C03605=1052.364,227.294,-95.651,172.051,36.072,156.780
C03606=1052.357,227.046,-95.623,172.050,36.069,156.779
C03607=1052.351,226.797,-95.597,172.047,36.065,156.779
C03608=1052.344,226.549,-95.569,172.045,36.062,156.778
C03609=1052.337,226.300,-95.542,172.042,36.058,156.777
C03610=1052.331,226.052,-95.515,172.040,36.055,156.777
C03611=1052.325,225.803,-95.488,172.038,36.052,156.776
C03612=1052.318,225.555,-95.460,172.036,36.048,156.775
C03613=1052.312,225.307,-95.434,172.034,36.045,156.775
C03614=1052.306,225.058,-95.406,172.032,36.042,156.774
C03615=1052.300,224.810,-95.379,172.029,36.038,156.773
C03616=1052.294,224.561,-95.352,172.027,36.035,156.772
C03617=1052.287,224.313,-95.326,172.026,36.032,156.772
C03618=1052.280,224.064,-95.299,172.023,36.028,156.771
C03619=1052.274,223.816,-95.271,172.021,36.024,156.770
C03620=1052.268,223.567,-95.244,172.018,36.021,156.770
C03621=1052.261,223.318,-95.217,172.016,36.018,156.769
C03622=1052.255,223.071,-95.190,172.015,36.014,156.768
C03623=1052.249,222.821,-95.163,172.012,36.011,156.768
C03624=1052.243,222.573,-95.137,172.010,36.007,156.767
C03625=1052.236,222.325,-95.109,172.008,36.004,156.766
C03626=1052.230,222.077,-95.082,172.005,36.000,156.765
C03627=1052.224,221.828,-95.055,172.004,35.997,156.765
C03628=1052.218,221.580,-95.028,172.001,35.993,156.764
C03629=1052.211,221.328,-95.001,171.999,35.990,156.763
C03630=1052.205,221.076,-94.974,171.997,35.987,156.763
C03631=1052.198,220.824,-94.946,171.995,35.983,156.762
C03632=1052.192,220.572,-94.919,171.993,35.979,156.761
C03633=1052.185,220.323,-94.893,171.991,35.976,156.760
C03634=1052.179,220.075,-94.865,171.988,35.973,156.760
C03635=1052.173,219.827,-94.839,171.987,35.969,156.759
C03636=1052.166,219.578,-94.812,171.985,35.966,156.758
C03637=1052.160,219.330,-94.786,171.982,35.963,156.758
C03638=1052.153,219.081,-94.759,171.980,35.959,156.757
C03639=1052.147,218.832,-94.733,171.977,35.956,156.756
C03640=1052.140,218.584,-94.706,171.976,35.953,156.756
C03641=1052.134,218.336,-94.679,171.974,35.949,156.755
C03642=1052.128,218.087,-94.652,171.971,35.945,156.754
C03643=1052.121,217.839,-94.626,171.970,35.942,156.753
C03644=1052.115,217.590,-94.599,171.968,35.939,156.753
C03645=1052.108,217.342,-94.573,171.965,35.935,156.752
C03646=1052.102,217.093,-94.546,171.963,35.932,156.751
C03647=1052.096,216.844,-94.519,171.962,35.929,156.751
C03648=1052.089,216.596,-94.493,171.959,35.925,156.750
C03649=1052.083,216.347,-94.466,171.957,35.921,156.749
C03650=1052.077,216.099,-94.440,171.955,35.918,156.749
C03651=1052.070,215.850,-94.413,171.953,35.915,156.748
C03652=1052.064,215.602,-94.387,171.951,35.911,156.747
C03653=1052.057,215.353,-94.360,171.949,35.908,156.746
C03654=1052.051,215.105,-94.334,171.947,35.904,156.746
C03655=1052.045,214.857,-94.307,171.945,35.900,156.745
C03656=1052.039,214.608,-94.280,171.942,35.897,156.744
C03657=1052.032,214.359,-94.254,171.941,35.894,156.744
C03658=1052.026,214.111,-94.227,171.939,35.890,156.743
C03659=1052.019,213.862,-94.201,171.936,35.887,156.742
C03660=1052.013,213.614,-94.174,171.934,35.883,156.741
C03661=1052.007,213.365,-94.149,171.933,35.880,156.741
C03662=1052.001,213.116,-94.122,171.930,35.876,156.740
C03663=1051.994,212.868,-94.096,171.928,35.873,156.739
C03664=1051.988,212.619,-94.069,171.927,35.869,156.739
C03665=1051.982,212.371,-94.043,171.924,35.865,156.738
C03666=1051.976,212.123,-94.016,171.922,35.862,156.737
C03667=1051.969,211.874,-93.990,171.921,35.859,156.737
C03668=1051.963,211.625,-93.964,171.918,35.855,156.736
C03669=1051.957,211.377,-93.938,171.916,35.852,156.735
C03670=1051.950,211.128,-93.911,171.914,35.848,156.734
C03671=1051.944,210.880,-93.885,171.912,35.845,156.734
C03672=1051.938,210.631,-93.859,171.910,35.841,156.733
C03673=1051.930,210.382,-93.833,171.908,35.838,156.732
C03674=1051.925,210.134,-93.806,171.906,35.834,156.732
C03675=1051.918,209.886,-93.780,171.905,35.831,156.731
C03676=1051.911,209.637,-93.755,171.902,35.828,156.730
C03677=1051.906,209.388,-93.728,171.900,35.824,156.730
C03678=1051.899,209.140,-93.702,171.899,35.820,156.729
C03679=1051.892,208.891,-93.676,171.896,35.817,156.728
C03680=1051.886,208.643,-93.650,171.894,35.813,156.727
C03681=1051.881,208.395,-93.624,171.893,35.810,156.727
C03682=1051.873,208.148,-93.598,171.890,35.807,156.726
C03683=1051.867,207.901,-93.572,171.888,35.803,156.725
C03684=1051.861,207.653,-93.546,171.887,35.799,156.725
C03685=1051.855,207.405,-93.520,171.884,35.796,156.724
C03686=1051.848,207.157,-93.494,171.883,35.793,156.723
C03687=1051.842,206.910,-93.469,171.881,35.789,156.722
C03688=1051.835,206.663,-93.442,171.878,35.785,156.722
C03689=1051.810,205.611,-93.337,171.657,35.690,156.704
C03690=1051.803,205.363,-93.312,171.654,35.688,156.704
C03691=1051.797,205.114,-93.287,171.652,35.686,156.703
C03692=1051.791,204.865,-93.262,171.649,35.683,156.703
C03693=1051.786,204.617,-93.237,171.647,35.680,156.702
C03694=1051.779,204.368,-93.212,171.644,35.678,156.702
C03695=1051.774,204.119,-93.187,171.642,35.675,156.701
C03696=1051.767,203.870,-93.162,171.639,35.672,156.701
C03697=1051.762,203.621,-93.138,171.637,35.669,156.700
C03698=1051.756,203.373,-93.112,171.634,35.667,156.699
C03699=1051.750,203.124,-93.087,171.632,35.664,156.699
C03700=1051.744,202.876,-93.063,171.629,35.661,156.698
C03701=1051.737,202.627,-93.038,171.626,35.659,156.698
C03702=1051.732,202.378,-93.013,171.624,35.656,156.697
C03703=1051.725,202.129,-92.988,171.622,35.653,156.697
C03704=1051.720,201.881,-92.964,171.619,35.651,156.696
C03705=1051.714,201.632,-92.938,171.617,35.648,156.696
C03706=1051.708,201.383,-92.914,171.614,35.645,156.695
C03707=1051.702,201.135,-92.889,171.612,35.643,156.695
C03708=1051.696,200.886,-92.865,171.609,35.640,156.694
C03709=1051.689,200.637,-92.840,171.606,35.638,156.694
C03710=1051.683,200.388,-92.815,171.604,35.635,156.693
C03711=1051.678,200.140,-92.791,171.602,35.633,156.693
C03712=1051.671,199.891,-92.766,171.600,35.630,156.692
C03713=1051.665,199.642,-92.742,171.596,35.627,156.692
C03714=1051.658,199.394,-92.717,171.594,35.625,156.691
C03715=1051.652,199.145,-92.693,171.592,35.622,156.691
C03716=1051.647,198.896,-92.668,171.590,35.620,156.690
C03717=1051.640,198.648,-92.644,171.586,35.617,156.690
C03718=1051.634,198.399,-92.619,171.584,35.614,156.689
C03719=1051.628,198.150,-92.595,171.582,35.612,156.689
C03720=1051.622,197.902,-92.570,171.580,35.610,156.688
C03721=1051.615,197.653,-92.546,171.578,35.607,156.688
C03722=1051.610,197.403,-92.521,171.574,35.605,156.687
C03723=1051.604,197.155,-92.497,171.572,35.602,156.687
C03724=1051.597,196.907,-92.472,171.570,35.600,156.687
C03725=1051.591,196.657,-92.448,171.568,35.597,156.686
C03726=1051.585,196.409,-92.424,171.564,35.594,156.685
C03727=1051.579,196.160,-92.400,171.562,35.592,156.685
C03728=1051.573,195.912,-92.375,171.560,35.589,156.684
C03729=1051.567,195.663,-92.351,171.558,35.587,156.684
C03730=1051.561,195.414,-92.326,171.556,35.584,156.684
C03731=1051.555,195.165,-92.302,171.552,35.582,156.683
C03732=1051.549,194.916,-92.278,171.550,35.579,156.683
C03733=1051.543,194.668,-92.253,171.548,35.577,156.682
C03734=1051.537,194.419,-92.229,171.546,35.574,156.682
C03735=1051.531,194.171,-92.205,171.543,35.571,156.681
C03736=1051.525,193.921,-92.180,171.541,35.569,156.681
C03737=1051.519,193.672,-92.156,171.538,35.566,156.680
C03738=1051.513,193.424,-92.132,171.536,35.564,156.680
C03739=1051.507,193.175,-92.108,171.534,35.562,156.679
C03740=1051.501,192.926,-92.084,171.531,35.559,156.679
C03741=1051.495,192.677,-92.060,171.529,35.557,156.678
C03742=1051.489,192.429,-92.035,171.527,35.554,156.678
C03743=1051.482,192.180,-92.011,171.524,35.552,156.677
C03744=1051.477,191.932,-91.986,171.522,35.549,156.677
C03745=1051.470,191.683,-91.962,171.519,35.547,156.676
C03746=1051.465,191.434,-91.938,171.517,35.544,156.676
C03747=1051.459,191.185,-91.914,171.515,35.542,156.675
C03748=1051.453,190.937,-91.890,171.513,35.539,156.675
C03749=1051.447,190.688,-91.866,171.509,35.536,156.674
C03750=1051.441,190.403,-91.838,171.507,35.534,156.674
C03751=1051.434,190.119,-91.810,171.505,35.531,156.673
C03752=1051.427,189.835,-91.783,171.502,35.528,156.673
C03753=1051.420,189.550,-91.756,171.500,35.525,156.672
C03754=1051.414,189.302,-91.732,171.497,35.523,156.672
C03755=1051.409,189.053,-91.708,171.494,35.520,156.671
C03756=1051.402,188.804,-91.684,171.492,35.518,156.671
C03757=1051.397,188.556,-91.660,171.490,35.515,156.670
C03758=1051.390,188.307,-91.636,171.487,35.513,156.670
C03759=1051.385,188.058,-91.611,171.485,35.510,156.669
C03760=1051.379,187.810,-91.588,171.483,35.508,156.669
C03761=1051.373,187.560,-91.563,171.481,35.505,156.668
C03762=1051.367,187.312,-91.540,171.479,35.502,156.668
C03763=1051.361,187.062,-91.516,171.476,35.500,156.667
C03764=1051.355,186.814,-91.492,171.473,35.497,156.667
C03765=1051.350,186.565,-91.468,171.471,35.495,156.666
C03766=1051.343,186.316,-91.444,171.469,35.492,156.666
C03767=1051.338,186.068,-91.419,171.467,35.490,156.665
C03768=1051.332,185.819,-91.396,171.464,35.487,156.665
C03769=1051.326,185.570,-91.372,171.462,35.485,156.665
C03770=1051.320,185.321,-91.348,171.460,35.483,156.664
C03771=1051.314,185.073,-91.324,171.458,35.480,156.664
C03772=1051.309,184.823,-91.301,171.456,35.478,156.663
C03773=1051.303,184.575,-91.277,171.453,35.475,156.663
C03774=1051.297,184.326,-91.253,171.451,35.473,156.662
C03775=1051.291,184.077,-91.229,171.449,35.470,156.662
C03776=1051.285,183.828,-91.206,171.446,35.468,156.661
C03777=1051.279,183.580,-91.182,171.444,35.466,156.661
C03778=1051.273,183.331,-91.159,171.441,35.463,156.660
C03779=1051.267,183.082,-91.135,171.439,35.461,156.660
C03780=1051.260,182.833,-91.111,171.437,35.458,156.659
C03781=1051.254,182.584,-91.088,171.435,35.457,156.659
C03782=1051.248,182.335,-91.064,171.433,35.454,156.659
C03783=1051.242,182.086,-91.041,171.430,35.452,156.658
C03784=1051.236,181.838,-91.017,171.428,35.450,156.658
C03785=1051.229,181.589,-90.994,171.425,35.447,156.657
C03786=1051.223,181.340,-90.970,171.423,35.445,156.657
C03787=1051.217,181.092,-90.948,171.421,35.442,156.656
C03788=1051.210,180.843,-90.924,171.419,35.440,156.656
C03789=1051.205,180.594,-90.901,171.416,35.438,156.656
C03790=1051.198,180.345,-90.877,171.414,35.435,156.655
C03791=1051.192,180.096,-90.854,171.412,35.434,156.655
C03792=1051.186,179.848,-90.830,171.410,35.431,156.654
C03793=1051.180,179.598,-90.807,171.408,35.429,156.654
C03794=1051.174,179.350,-90.783,171.405,35.426,156.653
C03795=1051.168,179.101,-90.761,171.403,35.424,156.653
C03796=1051.162,178.851,-90.737,171.401,35.422,156.653
C03797=1051.156,178.603,-90.714,171.399,35.419,156.652
C03798=1051.150,178.354,-90.691,171.396,35.417,156.652
C03799=1051.143,178.106,-90.667,171.394,35.415,156.651
C03800=1051.137,177.857,-90.644,171.391,35.412,156.651
C03801=1051.131,177.608,-90.621,171.389,35.411,156.650
C03802=1051.125,177.359,-90.598,171.387,35.408,156.650
C03803=1051.119,177.110,-90.574,171.385,35.406,156.649
C03804=1051.113,176.861,-90.551,171.383,35.404,156.649
C03805=1051.107,176.613,-90.528,171.380,35.401,156.649
C03806=1051.101,176.364,-90.505,171.378,35.399,156.648
C03807=1051.095,176.114,-90.481,171.376,35.396,156.648
C03808=1051.088,175.866,-90.458,171.374,35.394,156.647
C03809=1051.082,175.617,-90.435,171.372,35.392,156.647
C03810=1051.077,175.368,-90.413,171.370,35.389,156.646
C03811=1051.070,175.119,-90.389,171.367,35.388,156.646
C03812=1051.064,174.871,-90.366,171.365,35.385,156.646
C03813=1051.059,174.622,-90.343,171.363,35.383,156.645
C03814=1051.051,174.336,-90.317,171.361,35.380,156.645
C03815=1051.045,174.052,-90.290,171.358,35.378,156.644
C03816=1051.038,173.768,-90.264,171.355,35.375,156.644
C03817=1051.031,173.482,-90.237,171.353,35.372,156.643
C03818=1051.025,173.234,-90.214,171.351,35.370,156.643
C03819=1051.019,172.985,-90.191,171.349,35.368,156.642
C03820=1051.013,172.737,-90.168,171.347,35.365,156.642
C03821=1051.007,172.488,-90.145,171.344,35.363,156.642
C03822=1051.001,172.238,-90.122,171.342,35.361,156.641
C03823=1050.995,171.990,-90.098,171.340,35.358,156.641
C03824=1050.989,171.741,-90.075,171.338,35.357,156.640
C03825=1050.983,171.492,-90.052,171.336,35.354,156.640
C03826=1050.977,171.244,-90.030,171.334,35.352,156.639
C03827=1050.971,170.995,-90.007,171.331,35.350,156.639
C03828=1050.965,170.746,-89.984,171.329,35.347,156.639
C03829=1050.959,170.496,-89.961,171.327,35.345,156.638
C03830=1050.953,170.247,-89.938,171.325,35.343,156.638
C03831=1050.948,169.998,-89.915,171.323,35.340,156.637
C03832=1050.941,169.750,-89.893,171.321,35.338,156.637
C03833=1050.935,169.501,-89.870,171.318,35.336,156.636
C03834=1050.929,169.253,-89.846,171.316,35.333,156.636
C03835=1050.924,169.004,-89.823,171.314,35.331,156.635
C03836=1050.918,168.755,-89.800,171.312,35.329,156.635
C03837=1050.912,168.506,-89.777,171.310,35.327,156.635
C03838=1050.906,168.257,-89.755,171.307,35.324,156.634
C03839=1050.900,168.008,-89.732,171.305,35.322,156.634
C03840=1050.894,167.759,-89.709,171.303,35.320,156.633
C03841=1050.888,167.510,-89.686,171.301,35.317,156.633
C03842=1050.882,167.261,-89.663,171.299,35.315,156.633
C03843=1050.876,167.012,-89.641,171.297,35.313,156.632
C03844=1050.870,166.763,-89.618,171.294,35.310,156.632
C03845=1050.864,166.514,-89.595,171.292,35.309,156.631
C03846=1050.859,166.265,-89.572,171.291,35.306,156.631
C03847=1050.853,166.016,-89.549,171.289,35.304,156.630
C03848=1050.847,165.768,-89.527,171.287,35.302,156.630
C03849=1050.841,165.519,-89.504,171.285,35.299,156.630
C03850=1050.835,165.270,-89.481,171.282,35.297,156.629
C03851=1050.829,165.021,-89.458,171.280,35.295,156.629
C03852=1050.823,164.772,-89.436,171.278,35.292,156.628
C03853=1050.817,164.523,-89.413,171.276,35.290,156.628
C03854=1050.812,164.274,-89.391,171.274,35.288,156.627
C03855=1050.806,164.025,-89.368,171.272,35.285,156.627
C03856=1050.800,163.776,-89.345,171.269,35.283,156.627
C03857=1050.794,163.528,-89.322,171.267,35.281,156.626
C03858=1050.788,163.279,-89.299,171.265,35.279,156.626
C03859=1050.783,163.030,-89.277,171.264,35.276,156.625
C03860=1050.778,162.781,-89.255,171.262,35.274,156.625
C03861=1050.771,162.532,-89.232,171.260,35.272,156.624
C03862=1050.765,162.283,-89.209,171.257,35.269,156.624
C03863=1050.760,162.035,-89.186,171.255,35.267,156.624
C03864=1050.754,161.785,-89.164,171.253,35.265,156.623
C03865=1050.748,161.536,-89.142,171.251,35.263,156.623
C03866=1050.742,161.288,-89.119,171.249,35.260,156.622
C03867=1050.736,161.039,-89.096,171.247,35.258,156.622
C03868=1050.731,160.789,-89.074,171.245,35.256,156.622
C03869=1050.724,160.541,-89.051,171.243,35.254,156.621
C03870=1050.719,160.292,-89.028,171.241,35.252,156.621
C03871=1050.712,160.042,-89.007,171.239,35.249,156.620
C03872=1050.707,159.794,-88.984,171.237,35.247,156.620
C03873=1050.701,159.544,-88.962,171.235,35.245,156.619
C03874=1050.694,159.296,-88.940,171.232,35.243,156.619
C03875=1050.688,159.047,-88.917,171.230,35.240,156.619
C03876=1050.682,158.798,-88.895,171.228,35.239,156.618
C03877=1050.676,158.549,-88.873,171.226,35.236,156.618
C03878=1050.670,158.264,-88.847,171.224,35.234,156.617
C03879=1050.663,157.979,-88.822,171.222,35.231,156.617
C03880=1050.656,157.693,-88.796,171.219,35.229,156.616
C03881=1050.649,157.408,-88.771,171.217,35.227,156.616
C03882=1050.643,157.160,-88.749,171.215,35.224,156.616
C03883=1050.636,156.911,-88.727,171.213,35.222,156.615
C03884=1050.631,156.662,-88.704,171.211,35.220,156.615
C03885=1050.624,156.413,-88.682,171.209,35.218,156.614
C03886=1050.619,156.164,-88.660,171.207,35.215,156.614
C03887=1050.613,155.914,-88.638,171.204,35.214,156.614
C03888=1050.607,155.667,-88.616,171.202,35.211,156.613
C03889=1050.602,155.417,-88.594,171.201,35.209,156.613
C03890=1050.595,155.168,-88.572,171.199,35.207,156.612
C03891=1050.589,154.919,-88.550,171.197,35.205,156.612
C03892=1050.583,154.670,-88.527,171.195,35.203,156.612
C03893=1050.577,154.421,-88.505,171.192,35.200,156.611
C03894=1050.571,154.173,-88.483,171.190,35.198,156.611
C03895=1050.564,153.923,-88.461,171.188,35.196,156.610
C03896=1050.559,153.674,-88.439,171.187,35.194,156.610
C03897=1050.553,153.426,-88.417,171.185,35.192,156.610
C03898=1050.547,153.177,-88.396,171.183,35.190,156.609
C03899=1050.541,152.927,-88.374,171.181,35.188,156.609
C03900=1050.534,152.679,-88.352,171.178,35.185,156.608
C03901=1050.529,152.429,-88.329,171.176,35.183,156.608
C03902=1050.523,152.180,-88.308,171.174,35.182,156.608
C03903=1050.516,151.932,-88.285,171.172,35.179,156.607
C03904=1050.511,151.683,-88.264,171.171,35.177,156.607
C03905=1050.505,151.434,-88.242,171.169,35.175,156.607
C03906=1050.499,151.185,-88.219,171.167,35.173,156.606
C03907=1050.493,150.936,-88.198,171.164,35.171,156.606
C03908=1050.486,150.687,-88.176,171.162,35.168,156.605
C03909=1050.481,150.438,-88.155,171.160,35.166,156.605
C03910=1050.474,150.189,-88.133,171.159,35.165,156.605
C03911=1050.469,149.940,-88.110,171.157,35.162,156.604
C03912=1050.463,149.691,-88.089,171.155,35.160,156.604
C03913=1050.457,149.442,-88.067,171.152,35.158,156.603
C03914=1050.451,149.193,-88.046,171.150,35.156,156.603
C03915=1050.445,148.944,-88.023,171.148,35.154,156.603
C03916=1050.438,148.695,-88.002,171.147,35.151,156.602
C03917=1050.432,148.446,-87.980,171.145,35.150,156.602
C03918=1050.427,148.197,-87.958,171.143,35.148,156.602
C03919=1050.421,147.948,-87.937,171.141,35.145,156.601
C03920=1050.415,147.699,-87.914,171.138,35.143,156.601
C03921=1050.409,147.450,-87.893,171.136,35.141,156.600
C03922=1050.403,147.201,-87.871,171.135,35.139,156.600
C03923=1050.397,146.953,-87.850,171.133,35.137,156.600
C03924=1050.391,146.703,-87.828,171.131,35.135,156.599
C03925=1050.385,146.454,-87.807,171.129,35.133,156.599
C03926=1050.378,146.205,-87.785,171.127,35.131,156.598
C03927=1050.372,145.956,-87.763,171.125,35.129,156.598
C03928=1050.367,145.707,-87.742,171.123,35.126,156.598
C03929=1050.361,145.458,-87.720,171.121,35.124,156.597
C03930=1050.354,145.209,-87.699,171.119,35.122,156.597
C03931=1050.348,144.960,-87.678,171.117,35.121,156.597
C03932=1050.342,144.711,-87.656,171.115,35.118,156.596
C03933=1050.336,144.462,-87.635,171.113,35.116,156.596
C03934=1050.330,144.213,-87.613,171.112,35.114,156.596
C03935=1050.323,143.964,-87.592,171.109,35.112,156.595
C03936=1050.318,143.715,-87.570,171.107,35.110,156.595
C03937=1050.312,143.466,-87.549,171.105,35.108,156.594
C03938=1050.306,143.217,-87.527,171.103,35.106,156.594
C03939=1050.300,142.968,-87.506,171.102,35.104,156.594
C03940=1050.294,142.719,-87.484,171.100,35.102,156.593
C03941=1050.288,142.470,-87.462,171.098,35.100,156.593
C03942=1050.278,142.054,-87.427,171.094,35.096,156.592
C03943=1050.267,141.639,-87.391,171.091,35.093,156.592
C03944=1050.258,141.223,-87.356,171.088,35.089,156.591
C03945=1050.247,140.807,-87.320,171.085,35.086,156.590
C03946=1050.241,140.558,-87.298,171.082,35.083,156.590
C03947=1050.236,140.309,-87.277,171.080,35.081,156.590
C03948=1050.229,140.060,-87.255,171.079,35.080,156.589
C03949=1050.223,139.811,-87.234,171.077,35.077,156.589
C03950=1050.218,139.562,-87.213,171.075,35.075,156.588
C03951=1050.212,139.313,-87.191,171.073,35.073,156.588
C03952=1050.205,139.064,-87.170,171.072,35.071,156.588
C03953=1050.199,138.815,-87.149,171.070,35.070,156.587
C03954=1050.193,138.566,-87.128,171.067,35.067,156.587
C03955=1050.187,138.316,-87.107,171.065,35.065,156.587
C03956=1050.182,138.068,-87.085,171.063,35.063,156.586
C03957=1050.175,137.819,-87.064,171.062,35.061,156.586
C03958=1050.169,137.570,-87.043,171.060,35.059,156.585
C03959=1050.164,137.320,-87.022,171.058,35.057,156.585
C03960=1050.157,137.071,-87.000,171.056,35.055,156.585
C03961=1050.151,136.823,-86.980,171.055,35.053,156.584
C03962=1050.145,136.574,-86.958,171.052,35.051,156.584
C03963=1050.139,136.324,-86.937,171.050,35.049,156.584
C03964=1050.133,136.076,-86.917,171.048,35.047,156.583
C03965=1050.127,135.827,-86.895,171.046,35.045,156.583
C03966=1050.121,135.578,-86.874,171.045,35.043,156.583
C03967=1050.114,135.329,-86.853,171.043,35.040,156.582
C03968=1050.108,135.079,-86.832,171.041,35.039,156.582
C03969=1050.103,134.830,-86.811,171.038,35.037,156.581
C03970=1050.094,134.463,-86.779,171.036,35.034,156.581
C03971=1050.085,134.095,-86.749,171.033,35.031,156.580
C03972=1050.076,133.727,-86.718,171.031,35.028,156.580
C03973=1050.067,133.359,-86.687,171.028,35.025,156.579
C03974=1050.061,133.111,-86.666,171.026,35.023,156.579
C03975=1050.055,132.861,-86.645,171.024,35.021,156.579
C03976=1050.049,132.612,-86.624,171.022,35.018,156.578
C03977=1050.043,132.363,-86.604,171.020,35.016,156.578
C03978=1050.037,132.114,-86.582,171.018,35.015,156.577
C03979=1050.031,131.865,-86.561,171.017,35.013,156.577
C03980=1050.025,131.616,-86.540,171.015,35.011,156.577
C03981=1050.019,131.367,-86.520,171.013,35.008,156.576
C03982=1050.012,131.118,-86.499,171.011,35.006,156.576
C03983=1050.007,130.868,-86.478,171.009,35.004,156.576
C03984=1050.000,130.620,-86.457,171.007,35.003,156.575
C03985=1049.994,130.371,-86.437,171.005,35.001,156.575
C03986=1049.988,130.122,-86.416,171.003,34.999,156.575
C03987=1049.982,129.873,-86.395,171.002,34.997,156.574
C03988=1049.975,129.624,-86.375,171.000,34.995,156.574
C03989=1049.969,129.375,-86.354,170.998,34.993,156.574
C03990=1049.963,129.125,-86.333,170.996,34.991,156.573
C03991=1049.957,128.876,-86.312,170.994,34.989,156.573
C03992=1049.951,128.627,-86.292,170.992,34.987,156.572
C03993=1049.944,128.379,-86.271,170.990,34.985,156.572
C03994=1049.938,128.129,-86.250,170.988,34.983,156.572
C03995=1049.932,127.880,-86.230,170.987,34.981,156.571
C03996=1049.926,127.631,-86.209,170.985,34.979,156.571
C03997=1049.920,127.382,-86.189,170.983,34.977,156.571
C03998=1049.914,127.133,-86.168,170.981,34.975,156.570
C03999=1049.907,126.884,-86.148,170.980,34.973,156.570
C04000=1049.902,126.635,-86.127,170.977,34.971,156.570
C04001=1049.896,126.386,-86.107,170.975,34.970,156.569
C04002=1049.889,126.100,-86.083,170.973,34.967,156.569
C04003=1049.881,125.814,-86.059,170.971,34.965,156.569
C04004=1049.874,125.529,-86.035,170.969,34.963,156.568
C04005=1049.867,125.243,-86.012,170.967,34.960,156.568
C04006=1049.862,124.994,-85.991,170.965,34.958,156.567
C04007=1049.855,124.745,-85.971,170.963,34.956,156.567
C04008=1049.849,124.496,-85.951,170.961,34.954,156.567
C04009=1049.843,124.247,-85.929,170.959,34.952,156.566
C04010=1049.837,123.998,-85.909,170.958,34.951,156.566
C04011=1049.830,123.749,-85.889,170.956,34.949,156.566
C04012=1049.825,123.499,-85.868,170.954,34.947,156.565
C04013=1049.819,123.251,-85.848,170.952,34.945,156.565
C04014=1049.812,123.002,-85.827,170.951,34.943,156.565
C04015=1049.807,122.753,-85.807,170.949,34.940,156.564
C04016=1049.800,122.503,-85.787,170.946,34.938,156.564
C04017=1049.794,122.254,-85.767,170.945,34.937,156.564
C04018=1049.788,122.005,-85.746,170.943,34.935,156.563
C04019=1049.782,121.756,-85.725,170.941,34.933,156.563
C04020=1049.776,121.507,-85.705,170.939,34.931,156.563
C04021=1049.770,121.258,-85.685,170.938,34.929,156.562
C04022=1049.764,121.009,-85.664,170.936,34.927,156.562
C04023=1049.758,120.760,-85.644,170.934,34.924,156.561
C04024=1049.752,120.510,-85.624,170.932,34.923,156.561
C04025=1049.746,120.261,-85.603,170.930,34.921,156.561
C04026=1049.740,120.012,-85.582,170.928,34.919,156.560
C04027=1049.734,119.764,-85.562,170.927,34.917,156.560
C04028=1049.728,119.514,-85.542,170.925,34.915,156.560
C04029=1049.722,119.265,-85.521,170.923,34.913,156.559
C04030=1049.716,119.016,-85.501,170.922,34.911,156.559
C04031=1049.710,118.767,-85.482,170.920,34.909,156.559
C04032=1049.704,118.518,-85.461,170.918,34.907,156.558
C04033=1049.698,118.269,-85.441,170.915,34.905,156.558
C04034=1049.692,118.020,-85.421,170.914,34.903,156.558
C04035=1049.686,117.770,-85.400,170.912,34.901,156.557
C04036=1049.680,117.521,-85.380,170.910,34.899,156.557
C04037=1049.674,117.272,-85.360,170.909,34.897,156.556
C04038=1049.667,117.023,-85.340,170.907,34.895,156.556
C04039=1049.662,116.774,-85.319,170.905,34.893,156.556
C04040=1049.656,116.525,-85.299,170.904,34.891,156.555
C04041=1049.650,116.275,-85.279,170.902,34.889,156.555
C04042=1049.644,116.027,-85.259,170.899,34.887,156.555
C04043=1049.638,115.778,-85.238,170.898,34.885,156.554
C04044=1049.632,115.529,-85.218,170.896,34.883,156.554
C04045=1049.626,115.279,-85.198,170.894,34.881,156.554
C04046=1049.620,115.030,-85.178,170.893,34.879,156.553
C04047=1049.615,114.781,-85.157,170.891,34.877,156.553
C04048=1049.609,114.532,-85.137,170.889,34.875,156.553
C04049=1049.602,114.283,-85.117,170.888,34.873,156.552
C04050=1049.597,114.034,-85.097,170.885,34.870,156.552
C04051=1049.591,113.785,-85.077,170.883,34.869,156.551
C04052=1049.584,113.535,-85.057,170.882,34.867,156.551
C04053=1049.578,113.286,-85.037,170.880,34.865,156.551
C04054=1049.572,113.037,-85.017,170.878,34.863,156.550
C04055=1049.566,112.788,-84.997,170.877,34.861,156.550
C04056=1049.560,112.539,-84.977,170.875,34.859,156.550
C04057=1049.554,112.290,-84.957,170.873,34.857,156.549
C04058=1049.548,112.041,-84.938,170.872,34.855,156.549
C04059=1049.542,111.791,-84.917,170.869,34.853,156.549
C04060=1049.536,111.542,-84.897,170.867,34.851,156.548
C04061=1049.530,111.294,-84.877,170.866,34.849,156.548
C04062=1049.524,111.045,-84.857,170.864,34.848,156.548
C04063=1049.517,110.795,-84.838,170.862,34.846,156.547
C04064=1049.511,110.546,-84.818,170.861,34.844,156.547
C04065=1049.505,110.297,-84.798,170.859,34.842,156.547
C04066=1049.498,110.011,-84.775,170.857,34.839,156.546
C04067=1049.491,109.725,-84.753,170.855,34.837,156.546
C04068=1049.484,109.440,-84.730,170.852,34.835,156.546
C04069=1049.477,109.154,-84.707,170.850,34.833,156.545
C04070=1049.470,108.905,-84.688,170.849,34.831,156.545
C04071=1049.464,108.656,-84.668,170.847,34.829,156.544
C04072=1049.458,108.406,-84.648,170.845,34.827,156.544
C04073=1049.452,108.157,-84.628,170.844,34.825,156.544
C04074=1049.446,107.908,-84.608,170.842,34.823,156.543
C04075=1049.440,107.659,-84.589,170.840,34.821,156.543
C04076=1049.434,107.409,-84.569,170.839,34.819,156.543
C04077=1049.427,107.160,-84.550,170.836,34.818,156.542
C04078=1049.421,106.912,-84.530,170.834,34.816,156.542
C04079=1049.415,106.663,-84.510,170.833,34.814,156.542
C04080=1049.410,106.413,-84.491,170.831,34.812,156.541
C04081=1049.403,106.164,-84.471,170.829,34.810,156.541
C04082=1049.397,105.915,-84.451,170.828,34.808,156.541
C04083=1049.391,105.666,-84.432,170.826,34.806,156.540
C04084=1049.385,105.417,-84.412,170.824,34.804,156.540
C04085=1049.379,105.168,-84.393,170.823,34.802,156.540
C04086=1049.372,104.918,-84.373,170.821,34.800,156.539
C04087=1049.367,104.669,-84.353,170.818,34.798,156.539
C04088=1049.361,104.420,-84.333,170.817,34.796,156.539
C04089=1049.354,104.171,-84.315,170.815,34.795,156.538
C04090=1049.348,103.922,-84.295,170.813,34.793,156.538
C04091=1049.343,103.672,-84.276,170.812,34.791,156.538
C04092=1049.337,103.424,-84.256,170.810,34.789,156.537
C04093=1049.330,103.174,-84.235,170.808,34.787,156.537
C04094=1049.324,102.925,-84.217,170.807,34.785,156.537
C04095=1049.318,102.676,-84.197,170.805,34.783,156.536
C04096=1049.312,102.427,-84.177,170.804,34.781,156.536
C04097=1049.306,102.177,-84.158,170.801,34.779,156.536
C04098=1049.300,101.929,-84.138,170.799,34.777,156.535
C04099=1049.294,101.679,-84.120,170.798,34.775,156.535
C04100=1049.288,101.431,-84.100,170.796,34.773,156.535
C04101=1049.281,101.180,-84.080,170.794,34.771,156.534
C04102=1049.275,100.932,-84.060,170.793,34.770,156.534
C04103=1049.270,100.682,-84.041,170.791,34.768,156.534
C04104=1049.263,100.433,-84.022,170.789,34.766,156.533
C04105=1049.257,100.184,-84.002,170.788,34.764,156.533
C04106=1049.251,99.935,-83.983,170.785,34.762,156.533
C04107=1049.245,99.686,-83.964,170.783,34.760,156.532
C04108=1049.239,99.436,-83.944,170.782,34.758,156.532
C04109=1049.232,99.187,-83.925,170.780,34.756,156.532
C04110=1049.226,98.938,-83.905,170.779,34.754,156.531
C04111=1049.220,98.689,-83.887,170.777,34.752,156.531
C04112=1049.214,98.440,-83.867,170.775,34.750,156.531
C04113=1049.207,98.191,-83.848,170.774,34.748,156.530
C04114=1049.202,97.942,-83.829,170.772,34.747,156.530
C04115=1049.196,97.692,-83.810,170.770,34.745,156.530
C04116=1049.190,97.443,-83.791,170.769,34.743,156.529
C04117=1049.183,97.194,-83.771,170.766,34.741,156.529
C04118=1049.177,96.945,-83.752,170.764,34.739,156.529
C04119=1049.171,96.695,-83.733,170.763,34.738,156.528
C04120=1049.164,96.447,-83.713,170.761,34.736,156.528
C04121=1049.158,96.197,-83.694,170.759,34.734,156.528
C04122=1049.152,95.948,-83.675,170.758,34.732,156.527
C04123=1049.146,95.699,-83.656,170.756,34.730,156.527
C04124=1049.140,95.450,-83.638,170.755,34.728,156.527
C04125=1049.134,95.201,-83.618,170.753,34.726,156.526
C04126=1049.128,94.951,-83.598,170.751,34.724,156.526
C04127=1049.122,94.702,-83.580,170.749,34.722,156.526
C04128=1049.116,94.453,-83.560,170.747,34.720,156.525
C04129=1049.109,94.204,-83.541,170.745,34.718,156.525
C04130=1049.102,93.918,-83.519,170.744,34.716,156.525
C04131=1049.095,93.633,-83.498,170.742,34.714,156.524
C04132=1049.088,93.347,-83.476,170.740,34.712,156.524
C04133=1049.081,93.061,-83.454,170.738,34.710,156.524
C04134=1049.075,92.811,-83.434,170.736,34.708,156.523
C04135=1049.069,92.562,-83.416,170.735,34.706,156.523
C04136=1049.063,92.313,-83.396,170.733,34.704,156.523
C04137=1049.057,92.064,-83.378,170.730,34.702,156.522
C04138=1049.051,91.814,-83.359,170.729,34.700,156.522
C04139=1049.044,91.565,-83.340,170.727,34.698,156.522
C04140=1049.039,91.316,-83.321,170.726,34.697,156.521
C04141=1049.032,91.067,-83.302,170.724,34.695,156.521
C04142=1049.026,90.818,-83.282,170.722,34.693,156.521
C04143=1049.020,90.569,-83.263,170.721,34.691,156.520
C04144=1049.014,90.319,-83.244,170.719,34.689,156.520
C04145=1049.008,90.070,-83.225,170.717,34.687,156.520
C04146=1049.001,89.821,-83.207,170.716,34.686,156.519
C04147=1048.996,89.572,-83.188,170.713,34.684,156.519
C04148=1048.989,89.323,-83.169,170.711,34.682,156.519
C04149=1048.983,89.073,-83.150,170.710,34.680,156.518
C04150=1048.976,88.824,-83.132,170.708,34.678,156.518
C04151=1048.971,88.575,-83.112,170.707,34.676,156.518
C04152=1048.964,88.326,-83.094,170.705,34.674,156.517
C04153=1048.958,88.077,-83.075,170.703,34.673,156.517
C04154=1048.952,87.827,-83.057,170.702,34.671,156.517
C04155=1048.946,87.577,-83.038,170.700,34.669,156.517
C04156=1048.940,87.328,-83.019,170.698,34.667,156.516
C04157=1048.934,87.080,-83.001,170.697,34.665,156.516
C04158=1048.927,86.831,-82.982,170.694,34.663,156.516
C04159=1048.922,86.581,-82.963,170.693,34.661,156.515
C04160=1048.915,86.332,-82.944,170.691,34.660,156.515
C04161=1048.909,86.083,-82.926,170.689,34.658,156.515
C04162=1048.902,85.834,-82.907,170.688,34.656,156.514
C04163=1048.897,85.585,-82.888,170.686,34.654,156.514
C04164=1048.890,85.335,-82.869,170.684,34.652,156.514
C04165=1048.884,85.086,-82.851,170.683,34.650,156.513
C04166=1048.878,84.837,-82.833,170.681,34.648,156.513
C04167=1048.872,84.587,-82.813,170.679,34.646,156.513
C04168=1048.866,84.338,-82.795,170.678,34.645,156.513
C04169=1048.859,84.089,-82.776,170.676,34.643,156.512
C04170=1048.853,83.840,-82.757,170.674,34.641,156.512
C04171=1048.847,83.590,-82.740,170.672,34.639,156.512
C04172=1048.842,83.341,-82.721,170.670,34.637,156.511
C04173=1048.835,83.092,-82.702,170.669,34.635,156.511
C04174=1048.829,82.843,-82.683,170.667,34.633,156.511
C04175=1048.822,82.594,-82.665,170.666,34.631,156.510
C04176=1048.817,82.344,-82.646,170.664,34.630,156.510
C04177=1048.811,82.095,-82.628,170.662,34.628,156.510
C04178=1048.804,81.846,-82.609,170.661,34.626,156.509
C04179=1048.798,81.597,-82.590,170.659,34.624,156.509
C04180=1048.792,81.348,-82.572,170.657,34.622,156.509
C04181=1048.786,81.098,-82.553,170.655,34.621,156.508
C04182=1048.780,80.849,-82.535,170.653,34.619,156.508
C04183=1048.774,80.600,-82.516,170.652,34.617,156.508
C04184=1048.768,80.350,-82.498,170.650,34.615,156.507
C04185=1048.761,80.101,-82.480,170.648,34.613,156.507
C04186=1048.755,79.853,-82.461,170.647,34.611,156.507
C04187=1048.750,79.603,-82.442,170.645,34.609,156.506
C04188=1048.743,79.353,-82.424,170.644,34.608,156.506
C04189=1048.737,79.104,-82.405,170.642,34.606,156.506
C04190=1048.731,78.855,-82.387,170.640,34.604,156.505
C04191=1048.724,78.605,-82.369,170.639,34.602,156.505
C04192=1048.719,78.357,-82.351,170.636,34.600,156.505
C04193=1048.712,78.108,-82.332,170.634,34.598,156.504
C04194=1048.705,77.821,-82.311,170.633,34.596,156.504
C04195=1048.699,77.535,-82.290,170.631,34.594,156.504
C04196=1048.692,77.250,-82.269,170.629,34.591,156.503
C04197=1048.684,76.964,-82.248,170.627,34.590,156.503
C04198=1048.678,76.716,-82.230,170.625,34.588,156.503
C04199=1048.672,76.466,-82.212,170.624,34.586,156.502
C04200=1048.665,76.217,-82.193,170.622,34.584,156.502
C04201=1048.659,75.967,-82.175,170.621,34.582,156.502
C04202=1048.653,75.718,-82.157,170.619,34.580,156.501
C04203=1048.647,75.468,-82.139,170.617,34.579,156.501
C04204=1048.641,75.220,-82.120,170.615,34.577,156.501
C04205=1048.635,74.970,-82.102,170.613,34.575,156.501
C04206=1048.628,74.721,-82.084,170.611,34.573,156.500
C04207=1048.622,74.471,-82.066,170.610,34.571,156.500
C04208=1048.616,74.222,-82.047,170.608,34.569,156.500
C04209=1048.610,73.973,-82.030,170.607,34.568,156.499
C04210=1048.604,73.724,-82.011,170.605,34.566,156.499
C04211=1048.598,73.474,-81.993,170.603,34.564,156.499
C04212=1048.591,73.225,-81.974,170.602,34.562,156.498
C04213=1048.585,72.976,-81.957,170.600,34.560,156.498
C04214=1048.579,72.727,-81.939,170.598,34.558,156.498
C04215=1048.572,72.477,-81.921,170.597,34.557,156.497
C04216=1048.566,72.228,-81.902,170.594,34.555,156.497
C04217=1048.561,71.979,-81.885,170.593,34.553,156.497
C04218=1048.554,71.730,-81.866,170.591,34.551,156.497
C04219=1048.548,71.480,-81.848,170.589,34.549,156.496
C04220=1048.542,71.231,-81.830,170.588,34.548,156.496
C04221=1048.536,70.982,-81.812,170.586,34.546,156.496
C04222=1048.530,70.732,-81.794,170.584,34.544,156.495
C04223=1048.523,70.483,-81.777,170.583,34.542,156.495
C04224=1048.517,70.235,-81.758,170.581,34.540,156.495
C04225=1048.511,69.985,-81.740,170.580,34.538,156.494
C04226=1048.505,69.736,-81.722,170.578,34.536,156.494
C04227=1048.499,69.486,-81.704,170.576,34.535,156.494
C04228=1048.493,69.237,-81.686,170.575,34.533,156.493
C04229=1048.486,68.988,-81.668,170.572,34.531,156.493
C04230=1048.480,68.738,-81.650,170.570,34.529,156.493
C04231=1048.474,68.489,-81.632,170.569,34.527,156.492
C04232=1048.468,68.240,-81.615,170.567,34.526,156.492
C04233=1048.461,67.991,-81.597,170.566,34.524,156.492
C04234=1048.455,67.741,-81.579,170.564,34.522,156.492
C04235=1048.449,67.492,-81.561,170.562,34.520,156.491
C04236=1048.443,67.243,-81.543,170.561,34.519,156.491
C04237=1048.436,66.993,-81.525,170.559,34.517,156.491
C04238=1048.431,66.744,-81.508,170.557,34.515,156.490
C04239=1048.424,66.495,-81.490,170.556,34.513,156.490
C04240=1048.418,66.245,-81.471,170.554,34.511,156.490
C04241=1048.412,65.997,-81.454,170.553,34.510,156.490
C04242=1048.406,65.747,-81.436,170.550,34.508,156.489
C04243=1048.399,65.497,-81.418,170.548,34.506,156.489
C04244=1048.393,65.249,-81.401,170.547,34.504,156.489
C04245=1048.387,64.999,-81.383,170.545,34.503,156.488
C04246=1048.381,64.750,-81.365,170.543,34.501,156.488
C04247=1048.374,64.500,-81.347,170.542,34.499,156.488
C04248=1048.368,64.251,-81.330,170.540,34.497,156.487
C04249=1048.362,64.001,-81.312,170.539,34.496,156.487
C04250=1048.355,63.752,-81.294,170.537,34.494,156.487
C04251=1048.350,63.503,-81.277,170.535,34.492,156.486
C04252=1048.343,63.254,-81.260,170.534,34.490,156.486
C04253=1048.337,63.004,-81.241,170.532,34.488,156.486
C04254=1048.330,62.756,-81.224,170.530,34.486,156.486
C04255=1048.324,62.506,-81.206,170.528,34.485,156.485
C04256=1048.317,62.257,-81.189,170.526,34.483,156.485
C04257=1048.311,62.008,-81.172,170.524,34.481,156.485
C04258=1048.303,61.721,-81.151,170.523,34.479,156.484
C04259=1048.297,61.435,-81.131,170.521,34.477,156.484
C04260=1048.290,61.149,-81.112,170.519,34.475,156.484
C04261=1048.283,60.863,-81.092,170.517,34.473,156.483
C04262=1048.276,60.614,-81.074,170.515,34.472,156.483
C04263=1048.270,60.364,-81.056,170.514,34.470,156.483
C04264=1048.263,60.115,-81.039,170.512,34.468,156.483
C04265=1048.257,59.866,-81.021,170.510,34.467,156.482
C04266=1048.250,59.616,-81.004,170.509,34.465,156.482
C04267=1048.244,59.368,-80.987,170.507,34.463,156.482
C04268=1048.238,59.118,-80.969,170.505,34.462,156.481
C04269=1048.231,58.868,-80.952,170.503,34.460,156.481
C04270=1048.226,58.619,-80.934,170.501,34.458,156.481
C04271=1048.219,58.370,-80.917,170.499,34.456,156.481
C04272=1048.212,58.121,-80.900,170.498,34.454,156.480
C04273=1048.206,57.871,-80.882,170.496,34.453,156.480
C04274=1048.200,57.623,-80.865,170.494,34.451,156.480
C04275=1048.194,57.373,-80.847,170.493,34.449,156.479
C04276=1048.187,57.124,-80.830,170.491,34.447,156.479
C04277=1048.181,56.875,-80.813,170.490,34.446,156.479
C04278=1048.175,56.625,-80.795,170.488,34.444,156.479
C04279=1048.169,56.376,-80.778,170.486,34.442,156.478
C04280=1048.163,56.126,-80.761,170.485,34.441,156.478
C04281=1048.156,55.877,-80.744,170.483,34.439,156.478
C04282=1048.150,55.628,-80.726,170.481,34.437,156.477
C04283=1048.143,55.378,-80.708,170.480,34.436,156.477
C04284=1048.137,55.129,-80.691,170.477,34.434,156.477
C04285=1048.131,54.880,-80.673,170.475,34.432,156.477
C04286=1048.125,54.631,-80.657,170.474,34.430,156.476
C04287=1048.118,54.381,-80.640,170.472,34.428,156.476
C04288=1048.113,54.132,-80.622,170.470,34.426,156.476
C04289=1048.106,53.882,-80.605,170.469,34.424,156.475
C04290=1048.100,53.633,-80.587,170.467,34.423,156.475
C04291=1048.094,53.384,-80.570,170.466,34.421,156.475
C04292=1048.088,53.135,-80.554,170.464,34.419,156.474
C04293=1048.081,52.885,-80.536,170.462,34.418,156.474
C04294=1048.075,52.636,-80.519,170.461,34.416,156.474
C04295=1048.068,52.387,-80.502,170.459,34.414,156.474
C04296=1048.063,52.138,-80.484,170.457,34.413,156.473
C04297=1048.056,51.888,-80.467,170.456,34.411,156.473
C04298=1048.050,51.639,-80.450,170.453,34.409,156.473
C04299=1048.044,51.389,-80.432,170.451,34.407,156.472
C04300=1048.038,51.140,-80.416,170.450,34.405,156.472
C04301=1048.032,50.890,-80.398,170.448,34.403,156.472
C04302=1048.026,50.641,-80.381,170.447,34.402,156.472
C04303=1048.019,50.392,-80.364,170.445,34.400,156.471
C04304=1048.013,50.142,-80.347,170.443,34.398,156.471
C04305=1048.007,49.893,-80.330,170.442,34.396,156.471
C04306=1048.000,49.644,-80.313,170.440,34.394,156.470
C04307=1047.995,49.394,-80.296,170.438,34.393,156.470
C04308=1047.988,49.145,-80.279,170.437,34.391,156.470
C04309=1047.982,48.896,-80.262,170.435,34.389,156.469
C04310=1047.976,48.646,-80.244,170.433,34.388,156.469
C04311=1047.970,48.397,-80.227,170.432,34.386,156.469
C04312=1047.964,48.148,-80.211,170.430,34.384,156.469
C04313=1047.958,47.898,-80.193,170.428,34.382,156.468
C04314=1047.952,47.649,-80.176,170.426,34.381,156.468
C04315=1047.945,47.400,-80.159,170.424,34.379,156.468
C04316=1047.940,47.150,-80.142,170.423,34.377,156.467
C04317=1047.933,46.901,-80.125,170.421,34.375,156.467
C04318=1047.927,46.651,-80.109,170.419,34.373,156.467
C04319=1047.921,46.402,-80.091,170.418,34.371,156.467
C04320=1047.915,46.154,-80.074,170.416,34.370,156.466
C04321=1047.908,45.904,-80.057,170.414,34.368,156.466
C04322=1047.901,45.618,-80.037,170.413,34.366,156.466
C04323=1047.895,45.331,-80.018,170.411,34.364,156.465
C04324=1047.888,45.045,-79.998,170.409,34.362,156.465
C04325=1047.880,44.759,-79.980,170.407,34.360,156.465
C04326=1047.874,44.509,-79.962,170.405,34.358,156.464
C04327=1047.868,44.260,-79.945,170.404,34.356,156.464
C04328=1047.862,44.011,-79.928,170.401,34.354,156.464
C04329=1047.856,43.761,-79.911,170.399,34.352,156.463
C04330=1047.850,43.512,-79.894,170.398,34.351,156.463
C04331=1047.844,43.263,-79.878,170.396,34.349,156.463
C04332=1047.838,43.013,-79.861,170.394,34.347,156.463
C04333=1047.831,42.764,-79.844,170.393,34.345,156.462
C04334=1047.825,42.515,-79.828,170.391,34.344,156.462
C04335=1047.818,42.265,-79.811,170.389,34.342,156.462
C04336=1047.813,42.015,-79.794,170.388,34.341,156.462
C04337=1047.806,41.766,-79.777,170.386,34.339,156.461
C04338=1047.800,41.517,-79.760,170.384,34.337,156.461
C04339=1047.795,41.267,-79.744,170.383,34.335,156.461
C04340=1047.788,41.018,-79.727,170.381,34.333,156.460
C04341=1047.782,40.769,-79.710,170.379,34.331,156.460
C04342=1047.775,40.520,-79.694,170.378,34.330,156.460
C04343=1047.769,40.270,-79.677,170.376,34.328,156.459
C04344=1047.763,40.020,-79.661,170.374,34.327,156.459
C04345=1047.757,39.772,-79.644,170.372,34.325,156.459
C04346=1047.751,39.522,-79.627,170.370,34.323,156.459
C04347=1047.744,39.272,-79.611,170.368,34.322,156.458
C04348=1047.738,39.024,-79.594,170.367,34.320,156.458
C04349=1047.732,38.774,-79.578,170.365,34.318,156.458
C04350=1047.725,38.524,-79.561,170.363,34.316,156.458
C04351=1047.719,38.275,-79.544,170.362,34.314,156.457
C04352=1047.713,38.026,-79.528,170.360,34.313,156.457
C04353=1047.707,37.777,-79.511,170.358,34.311,156.457
C04354=1047.701,37.527,-79.495,170.357,34.309,156.456
C04355=1047.694,37.278,-79.478,170.355,34.308,156.456
C04356=1047.689,37.029,-79.462,170.353,34.306,156.456
C04357=1047.682,36.779,-79.445,170.352,34.304,156.456
C04358=1047.676,36.529,-79.429,170.350,34.302,156.455
C04359=1047.670,36.281,-79.412,170.348,34.301,156.455
C04360=1047.663,36.030,-79.395,170.347,34.299,156.455
C04361=1047.656,35.781,-79.379,170.345,34.298,156.455
C04362=1047.651,35.532,-79.363,170.342,34.296,156.454
C04363=1047.645,35.283,-79.347,170.341,34.295,156.454
C04364=1047.638,35.033,-79.330,170.339,34.293,156.454
C04365=1047.632,34.784,-79.313,170.337,34.291,156.454
C04366=1047.626,34.535,-79.297,170.335,34.289,156.453
C04367=1047.619,34.285,-79.281,170.334,34.288,156.453
C04368=1047.613,34.036,-79.265,170.332,34.286,156.453
C04369=1047.607,33.786,-79.249,170.330,34.284,156.452
C04370=1047.600,33.537,-79.232,170.329,34.283,156.452
C04371=1047.594,33.287,-79.215,170.327,34.281,156.452
C04372=1047.587,33.038,-79.199,170.325,34.279,156.452
C04373=1047.581,32.789,-79.183,170.324,34.277,156.451
C04374=1047.575,32.540,-79.167,170.322,34.276,156.451
C04375=1047.569,32.290,-79.151,170.320,34.274,156.451
C04376=1047.563,32.040,-79.134,170.319,34.273,156.451
C04377=1047.557,31.791,-79.118,170.317,34.271,156.450
C04378=1047.550,31.542,-79.102,170.315,34.269,156.450
C04379=1047.544,31.293,-79.086,170.314,34.267,156.450
C04380=1047.538,31.042,-79.069,170.312,34.266,156.449
C04381=1047.531,30.794,-79.052,170.309,34.264,156.449
C04382=1047.525,30.544,-79.036,170.307,34.263,156.449
C04383=1047.519,30.295,-79.020,170.306,34.261,156.449
C04384=1047.513,30.046,-79.004,170.304,34.259,156.448
C04385=1047.507,29.797,-78.988,170.302,34.257,156.448
C04386=1047.500,29.510,-78.970,170.300,34.255,156.448
C04387=1047.492,29.224,-78.951,170.298,34.253,156.447
C04388=1047.486,28.937,-78.932,170.297,34.252,156.447
C04389=1047.478,28.651,-78.913,170.295,34.250,156.447
C04390=1047.472,28.402,-78.898,170.293,34.248,156.447
C04391=1047.466,28.152,-78.881,170.291,34.246,156.446
C04392=1047.459,27.902,-78.865,170.289,34.245,156.446
C04393=1047.452,27.653,-78.849,170.288,34.243,156.446
C04394=1047.446,27.404,-78.833,170.286,34.242,156.446
C04395=1047.440,27.155,-78.817,170.284,34.240,156.445
C04396=1047.434,26.905,-78.802,170.283,34.238,156.445
C04397=1047.428,26.656,-78.785,170.281,34.236,156.445
C04398=1047.422,26.406,-78.769,170.279,34.235,156.445
C04399=1047.415,26.156,-78.753,170.278,34.234,156.444
C04400=1047.409,25.907,-78.737,170.275,34.232,156.444
C04401=1047.402,25.658,-78.721,170.273,34.230,156.444
C04402=1047.396,25.409,-78.705,170.271,34.228,156.443
C04403=1047.390,25.159,-78.689,170.270,34.227,156.443
C04404=1047.384,24.910,-78.674,170.268,34.225,156.443
C04405=1047.377,24.660,-78.657,170.266,34.224,156.443
C04406=1047.371,24.411,-78.641,170.264,34.222,156.442
C04407=1047.365,24.161,-78.625,170.263,34.220,156.442
C04408=1047.358,23.912,-78.609,170.261,34.219,156.442
C04409=1047.352,23.662,-78.594,170.259,34.217,156.442
C04410=1047.346,23.413,-78.578,170.258,34.216,156.441
C04411=1047.340,23.164,-78.562,170.256,34.214,156.441
C04412=1047.334,22.915,-78.546,170.254,34.212,156.441
C04413=1047.327,22.666,-78.530,170.252,34.210,156.441
C04414=1047.321,22.415,-78.514,170.251,34.209,156.440
C04415=1047.314,22.166,-78.499,170.249,34.207,156.440
C04416=1047.308,21.916,-78.482,170.247,34.206,156.440
C04417=1047.302,21.667,-78.467,170.246,34.204,156.440
C04418=1047.296,21.417,-78.451,170.244,34.202,156.439
C04419=1047.290,21.168,-78.435,170.242,34.201,156.439
C04420=1047.283,20.919,-78.419,170.240,34.199,156.439
C04421=1047.277,20.670,-78.403,170.238,34.198,156.439
C04422=1047.271,20.420,-78.388,170.236,34.196,156.438
C04423=1047.265,20.171,-78.372,170.234,34.194,156.438
C04424=1047.258,19.922,-78.356,170.232,34.192,156.438
C04425=1047.253,19.672,-78.341,170.231,34.191,156.438
C04426=1047.246,19.423,-78.325,170.229,34.190,156.437
C04427=1047.239,19.174,-78.309,170.227,34.188,156.437
C04428=1047.234,18.924,-78.294,170.225,34.186,156.437
C04429=1047.226,18.674,-78.278,170.224,34.185,156.437
C04430=1047.221,18.424,-78.262,170.222,34.183,156.436
C04431=1047.214,18.175,-78.246,170.220,34.182,156.436
C04432=1047.208,17.926,-78.230,170.218,34.180,156.436
C04433=1047.202,17.676,-78.215,170.217,34.178,156.436
C04434=1047.195,17.427,-78.200,170.215,34.177,156.435
C04435=1047.189,17.177,-78.184,170.213,34.175,156.435
C04436=1047.183,16.928,-78.168,170.212,34.174,156.435
C04437=1047.177,16.679,-78.152,170.210,34.172,156.435
C04438=1047.170,16.429,-78.137,170.208,34.170,156.434
C04439=1047.164,16.180,-78.121,170.206,34.169,156.434
C04440=1047.158,15.930,-78.106,170.205,34.167,156.434
C04441=1047.151,15.681,-78.090,170.203,34.166,156.434
C04442=1047.146,15.431,-78.075,170.201,34.164,156.433
C04443=1047.139,15.182,-78.059,170.199,34.162,156.433
C04444=1047.133,14.932,-78.044,170.197,34.161,156.433
C04445=1047.127,14.683,-78.028,170.195,34.159,156.433
C04446=1047.120,14.433,-78.013,170.193,34.157,156.432
C04447=1047.114,14.184,-77.997,170.191,34.156,156.432
C04448=1047.108,13.934,-77.982,170.189,34.154,156.432
C04449=1047.101,13.685,-77.966,170.188,34.153,156.432
C04450=1047.094,13.401,-77.949,170.186,34.151,156.431
C04451=1047.087,13.115,-77.931,170.184,34.149,156.431
C04452=1047.079,12.830,-77.913,170.182,34.147,156.431
C04453=1047.073,12.545,-77.897,170.180,34.146,156.431
C04454=1047.066,12.296,-77.881,170.178,34.145,156.430
C04455=1047.060,12.046,-77.866,170.176,34.143,156.430
C04456=1047.053,11.797,-77.851,170.174,34.141,156.430
C04457=1047.047,11.547,-77.835,170.172,34.140,156.430
C04458=1047.041,11.298,-77.820,170.171,34.139,156.429
C04459=1047.034,11.049,-77.804,170.169,34.137,156.429
C04460=1047.028,10.799,-77.789,170.167,34.135,156.429
C04461=1047.021,10.549,-77.774,170.165,34.134,156.429
C04462=1047.015,10.300,-77.759,170.164,34.133,156.429
C04463=1047.008,10.051,-77.744,170.162,34.131,156.428
C04464=1047.003,9.801,-77.728,170.160,34.129,156.428
C04465=1046.996,9.552,-77.713,170.158,34.128,156.428
C04466=1046.990,9.302,-77.698,170.156,34.126,156.428
C04467=1046.983,9.052,-77.683,170.155,34.124,156.427
C04468=1046.977,8.803,-77.667,170.153,34.123,156.427
C04469=1046.970,8.554,-77.652,170.151,34.122,156.427
C04470=1046.964,8.304,-77.637,170.149,34.120,156.427
C04471=1046.957,8.054,-77.622,170.146,34.118,156.426
C04472=1046.952,7.806,-77.606,170.145,34.117,156.426
C04473=1046.946,7.556,-77.591,170.143,34.116,156.426
C04474=1046.939,7.306,-77.576,170.141,34.114,156.426
C04475=1046.933,7.057,-77.562,170.139,34.112,156.425
C04476=1046.926,6.808,-77.546,170.137,34.111,156.425
C04477=1046.920,6.558,-77.531,170.136,34.110,156.425
C04478=1046.913,6.308,-77.516,170.134,34.108,156.425
C04479=1046.907,6.059,-77.501,170.132,34.106,156.425
C04480=1046.901,5.810,-77.486,170.130,34.105,156.424
C04481=1046.895,5.561,-77.471,170.129,34.104,156.424
C04482=1046.889,5.311,-77.455,170.127,34.102,156.424
C04483=1046.883,5.061,-77.440,170.125,34.100,156.424
C04484=1046.876,4.811,-77.425,170.123,34.099,156.423
C04485=1046.870,4.562,-77.410,170.121,34.097,156.423
C04486=1046.863,4.313,-77.395,170.120,34.096,156.423
C04487=1046.857,4.064,-77.380,170.118,34.094,156.423
C04488=1046.851,3.814,-77.365,170.116,34.093,156.422
C04489=1046.845,3.564,-77.350,170.114,34.091,156.422
C04490=1046.838,3.315,-77.335,170.112,34.090,156.422
C04491=1046.832,3.065,-77.320,170.110,34.088,156.422
C04492=1046.826,2.816,-77.306,170.109,34.087,156.422
C04493=1046.820,2.566,-77.290,170.107,34.085,156.421
C04494=1046.814,2.317,-77.275,170.105,34.084,156.421
C04495=1046.807,2.068,-77.260,170.103,34.082,156.421
C04496=1046.801,1.818,-77.245,170.101,34.080,156.421
C04497=1046.795,1.569,-77.230,170.100,34.079,156.420
C04498=1046.789,1.319,-77.215,170.098,34.078,156.420
C04499=1046.782,1.070,-77.200,170.095,34.076,156.420
C04500=1046.776,0.820,-77.185,170.093,34.074,156.420
C04501=1046.770,0.571,-77.171,170.091,34.073,156.420
C04502=1046.764,0.321,-77.156,170.090,34.072,156.419
C04503=1046.757,0.072,-77.141,170.088,34.070,156.419
C04504=1046.751,-0.178,-77.126,170.086,34.068,156.419
C04505=1046.745,-0.427,-77.111,170.084,34.067,156.419
C04506=1046.739,-0.677,-77.096,170.082,34.066,156.418
C04507=1046.732,-0.926,-77.081,170.081,34.064,156.418
C04508=1046.726,-1.176,-77.066,170.079,34.062,156.418
C04509=1046.720,-1.425,-77.052,170.077,34.061,156.418
C04510=1046.714,-1.675,-77.037,170.075,34.059,156.417
C04511=1046.708,-1.924,-77.021,170.073,34.057,156.417
C04512=1046.702,-2.173,-77.007,170.071,34.056,156.417
C04513=1046.696,-2.423,-76.992,170.070,34.055,156.417
C04514=1046.689,-2.707,-76.976,170.068,34.053,156.416
C04515=1046.682,-2.989,-76.958,170.065,34.051,156.416
C04516=1046.675,-3.273,-76.942,170.063,34.049,156.416
C04517=1046.667,-3.556,-76.925,170.061,34.048,156.416
C04518=1046.661,-3.805,-76.910,170.059,34.046,156.416
C04519=1046.655,-4.054,-76.896,170.058,34.045,156.415
C04520=1046.649,-4.305,-76.881,170.056,34.044,156.415
C04521=1046.642,-4.554,-76.867,170.054,34.042,156.415
C04522=1046.636,-4.803,-76.852,170.052,34.041,156.415
C04523=1046.630,-5.053,-76.837,170.050,34.040,156.415
C04524=1046.623,-5.302,-76.822,170.048,34.038,156.414
C04525=1046.617,-5.552,-76.809,170.046,34.036,156.414
C04526=1046.611,-5.801,-76.794,170.045,34.035,156.414
C04527=1046.604,-6.051,-76.779,170.043,34.034,156.414
C04528=1046.598,-6.300,-76.764,170.041,34.032,156.413
C04529=1046.591,-6.549,-76.750,170.039,34.031,156.413
C04530=1046.585,-6.799,-76.736,170.037,34.029,156.413
C04531=1046.579,-7.049,-76.721,170.035,34.028,156.413
C04532=1046.572,-7.298,-76.707,170.033,34.027,156.413
C04533=1046.566,-7.547,-76.692,170.031,34.025,156.412
C04534=1046.560,-7.798,-76.678,170.029,34.024,156.412
C04535=1046.554,-8.047,-76.663,170.027,34.023,156.412
C04536=1046.547,-8.296,-76.649,170.025,34.021,156.412
C04537=1046.541,-8.546,-76.635,170.023,34.020,156.412
C04538=1046.535,-8.795,-76.620,170.021,34.018,156.411
C04539=1046.528,-9.045,-76.606,170.019,34.017,156.411
C04540=1046.522,-9.294,-76.591,170.017,34.016,156.411
C04541=1046.516,-9.544,-76.577,170.016,34.014,156.411
C04542=1046.510,-9.793,-76.562,170.014,34.013,156.411
C04543=1046.503,-10.042,-76.548,170.012,34.011,156.410
C04544=1046.497,-10.292,-76.534,170.010,34.009,156.410
C04545=1046.491,-10.542,-76.519,170.008,34.008,156.410
C04546=1046.484,-10.791,-76.505,170.006,34.007,156.410
C04547=1046.478,-11.041,-76.491,170.004,34.005,156.410
C04548=1046.472,-11.290,-76.476,170.002,34.004,156.409
C04549=1046.466,-11.540,-76.463,170.000,34.003,156.409
C04550=1046.459,-11.789,-76.448,169.999,34.001,156.409
C04551=1046.453,-12.038,-76.433,169.997,34.000,156.409
C04552=1046.447,-12.288,-76.419,169.995,33.998,156.409
C04553=1046.441,-12.537,-76.405,169.993,33.997,156.408
C04554=1046.435,-12.788,-76.391,169.991,33.996,156.408
C04555=1046.428,-13.037,-76.376,169.989,33.994,156.408
C04556=1046.422,-13.287,-76.362,169.987,33.993,156.408
C04557=1046.416,-13.536,-76.347,169.985,33.991,156.408
C04558=1046.409,-13.785,-76.333,169.984,33.990,156.407
C04559=1046.403,-14.035,-76.319,169.982,33.989,156.407
C04560=1046.397,-14.284,-76.305,169.980,33.987,156.407
C04561=1046.391,-14.534,-76.291,169.978,33.986,156.407
C04562=1046.385,-14.783,-76.276,169.976,33.985,156.407
C04563=1046.379,-15.033,-76.262,169.974,33.983,156.406
C04564=1046.372,-15.282,-76.248,169.972,33.982,156.406
C04565=1046.366,-15.532,-76.234,169.970,33.980,156.406
C04566=1046.359,-15.782,-76.220,169.968,33.979,156.406
C04567=1046.354,-16.031,-76.206,169.966,33.978,156.406
C04568=1046.347,-16.281,-76.192,169.964,33.976,156.405
C04569=1046.341,-16.530,-76.178,169.963,33.975,156.405
C04570=1046.334,-16.780,-76.164,169.961,33.974,156.405
C04571=1046.328,-17.029,-76.150,169.959,33.973,156.405
C04572=1046.322,-17.279,-76.136,169.957,33.971,156.405
C04573=1046.315,-17.528,-76.122,169.955,33.970,156.405
C04574=1046.309,-17.778,-76.107,169.953,33.969,156.404
C04575=1046.302,-18.028,-76.094,169.951,33.967,156.404
C04576=1046.296,-18.277,-76.079,169.949,33.966,156.404
C04577=1046.290,-18.527,-76.066,169.947,33.964,156.404
C04578=1046.283,-18.808,-76.050,169.944,33.963,156.404
C04579=1046.276,-19.090,-76.035,169.942,33.962,156.403
C04580=1046.268,-19.371,-76.019,169.940,33.960,156.403
C04581=1046.262,-19.653,-76.003,169.937,33.959,156.403
C04582=1046.255,-19.902,-75.989,169.935,33.957,156.403
C04583=1046.249,-20.151,-75.975,169.934,33.956,156.403
C04584=1046.242,-20.401,-75.961,169.932,33.955,156.402
C04585=1046.237,-20.651,-75.947,169.930,33.953,156.402
C04586=1046.230,-20.900,-75.933,169.928,33.952,156.402
C04587=1046.223,-21.150,-75.920,169.926,33.951,156.402
C04588=1046.217,-21.400,-75.905,169.924,33.950,156.402
C04589=1046.211,-21.649,-75.892,169.922,33.948,156.401
C04590=1046.205,-21.898,-75.878,169.920,33.947,156.401
C04591=1046.198,-22.148,-75.864,169.918,33.946,156.401
C04592=1046.192,-22.397,-75.851,169.916,33.944,156.401
C04593=1046.186,-22.648,-75.836,169.914,33.943,156.401
C04594=1046.180,-22.896,-75.823,169.912,33.941,156.401
C04595=1046.174,-23.147,-75.808,169.910,33.941,156.400
C04596=1046.167,-23.396,-75.795,169.908,33.939,156.400
C04597=1046.161,-23.645,-75.782,169.906,33.938,156.400
C04598=1046.155,-23.895,-75.768,169.904,33.936,156.400
C04599=1046.149,-24.144,-75.754,169.902,33.935,156.400
C04600=1046.142,-24.394,-75.740,169.900,33.934,156.399
C04601=1046.136,-24.644,-75.726,169.899,33.932,156.399
C04602=1046.130,-24.893,-75.713,169.897,33.932,156.399
C04603=1046.124,-25.143,-75.699,169.895,33.930,156.399
C04604=1046.118,-25.392,-75.685,169.893,33.929,156.399
C04605=1046.112,-25.642,-75.672,169.891,33.927,156.399
C04606=1046.105,-25.891,-75.657,169.889,33.926,156.398
C04607=1046.099,-26.140,-75.644,169.887,33.925,156.398
C04608=1046.092,-26.390,-75.630,169.885,33.924,156.398
C04609=1046.087,-26.640,-75.616,169.883,33.922,156.398
C04610=1046.080,-26.889,-75.603,169.881,33.921,156.398
C04611=1046.074,-27.139,-75.589,169.879,33.920,156.398
C04612=1046.067,-27.389,-75.576,169.877,33.918,156.397
C04613=1046.062,-27.638,-75.562,169.875,33.917,156.397
C04614=1046.055,-27.888,-75.549,169.873,33.916,156.397
C04615=1046.049,-28.137,-75.535,169.871,33.915,156.397
C04616=1046.042,-28.387,-75.522,169.869,33.914,156.397
C04617=1046.036,-28.637,-75.508,169.867,33.913,156.397
C04618=1046.030,-28.886,-75.495,169.865,33.911,156.396
C04619=1046.023,-29.136,-75.482,169.863,33.910,156.396
C04620=1046.017,-29.385,-75.468,169.861,33.909,156.396
C04621=1046.011,-29.635,-75.454,169.859,33.908,156.396
C04622=1046.004,-29.885,-75.441,169.857,33.907,156.396
C04623=1045.998,-30.134,-75.427,169.855,33.905,156.396
C04624=1045.992,-30.383,-75.414,169.853,33.904,156.395
C04625=1045.985,-30.633,-75.401,169.851,33.903,156.395
C04626=1045.979,-30.882,-75.387,169.849,33.902,156.395
C04627=1045.973,-31.132,-75.374,169.847,33.900,156.395
C04628=1045.966,-31.382,-75.360,169.845,33.900,156.395
C04629=1045.960,-31.631,-75.347,169.843,33.898,156.395
C04630=1045.954,-31.880,-75.333,169.841,33.897,156.395
C04631=1045.948,-32.130,-75.321,169.839,33.895,156.394
C04632=1045.941,-32.380,-75.307,169.837,33.895,156.394
C04633=1045.935,-32.630,-75.294,169.835,33.893,156.394
C04634=1045.929,-32.879,-75.281,169.833,33.893,156.394
C04635=1045.922,-33.129,-75.267,169.831,33.891,156.394
C04636=1045.916,-33.378,-75.254,169.829,33.890,156.394
C04637=1045.910,-33.627,-75.240,169.827,33.889,156.393
C04638=1045.904,-33.877,-75.228,169.825,33.888,156.393
C04639=1045.897,-34.127,-75.214,169.823,33.886,156.393
C04640=1045.891,-34.376,-75.201,169.821,33.885,156.393
C04641=1045.885,-34.626,-75.188,169.819,33.884,156.393
C04642=1045.878,-34.907,-75.172,169.817,33.883,156.393
C04643=1045.871,-35.187,-75.158,169.814,33.881,156.392
C04644=1045.864,-35.468,-75.143,169.812,33.880,156.392
C04645=1045.857,-35.749,-75.127,169.810,33.879,156.392
C04646=1045.851,-35.999,-75.115,169.808,33.878,156.392
C04647=1045.845,-36.248,-75.101,169.806,33.876,156.392
C04648=1045.838,-36.498,-75.088,169.804,33.875,156.392
C04649=1045.832,-36.747,-75.075,169.802,33.874,156.392
C04650=1045.826,-36.997,-75.062,169.800,33.873,156.391
C04651=1045.820,-37.246,-75.049,169.798,33.872,156.391
C04652=1045.813,-37.495,-75.035,169.796,33.870,156.391
C04653=1045.807,-37.745,-75.022,169.794,33.869,156.391
C04654=1045.801,-37.995,-75.009,169.792,33.868,156.391
C04655=1045.794,-38.245,-74.996,169.790,33.867,156.391
C04656=1045.788,-38.494,-74.983,169.788,33.866,156.391
C04657=1045.782,-38.744,-74.970,169.786,33.865,156.390
C04658=1045.776,-38.993,-74.957,169.783,33.863,156.390
C04659=1045.770,-39.244,-74.944,169.781,33.862,156.390
C04660=1045.763,-39.493,-74.931,169.779,33.862,156.390
C04661=1045.757,-39.742,-74.917,169.777,33.860,156.390
C04662=1045.751,-39.992,-74.905,169.775,33.859,156.390
C04663=1045.744,-40.241,-74.892,169.773,33.858,156.390
C04664=1045.738,-40.491,-74.879,169.771,33.857,156.389
C04665=1045.732,-40.741,-74.866,169.769,33.856,156.389
C04666=1045.725,-40.990,-74.853,169.767,33.855,156.389
C04667=1045.719,-41.240,-74.840,169.765,33.854,156.389
C04668=1045.713,-41.489,-74.828,169.763,33.853,156.389
C04669=1045.707,-41.739,-74.815,169.761,33.851,156.389
C04670=1045.700,-41.988,-74.802,169.759,33.851,156.389
C04671=1045.694,-42.239,-74.789,169.756,33.849,156.388
C04672=1045.688,-42.488,-74.776,169.754,33.849,156.388
C04673=1045.681,-42.737,-74.764,169.753,33.848,156.388
C04674=1045.675,-42.987,-74.750,169.750,33.846,156.388
C04675=1045.669,-43.237,-74.738,169.748,33.846,156.388
C04676=1045.663,-43.486,-74.724,169.745,33.844,156.388
C04677=1045.657,-43.736,-74.712,169.743,33.843,156.388
C04678=1045.650,-43.985,-74.699,169.741,33.842,156.388
C04679=1045.643,-44.235,-74.686,169.739,33.841,156.387
C04680=1045.637,-44.485,-74.673,169.737,33.840,156.387
C04681=1045.631,-44.734,-74.661,169.735,33.839,156.387
C04682=1045.625,-44.984,-74.647,169.733,33.838,156.387
C04683=1045.618,-45.233,-74.635,169.731,33.837,156.387
C04684=1045.612,-45.483,-74.622,169.729,33.836,156.387
C04685=1045.606,-45.732,-74.609,169.727,33.835,156.387
C04686=1045.600,-45.982,-74.597,169.725,33.834,156.387
C04687=1045.593,-46.231,-74.584,169.723,33.832,156.386
C04688=1045.587,-46.481,-74.572,169.720,33.832,156.386
C04689=1045.581,-46.730,-74.558,169.718,33.831,156.386
C04690=1045.575,-46.980,-74.546,169.716,33.829,156.386
C04691=1045.569,-47.230,-74.533,169.714,33.829,156.386
C04692=1045.562,-47.479,-74.521,169.712,33.827,156.386
C04693=1045.557,-47.729,-74.508,169.710,33.826,156.386
C04694=1045.550,-47.978,-74.495,169.708,33.826,156.386
C04695=1045.544,-48.228,-74.482,169.706,33.824,156.385
C04696=1045.538,-48.478,-74.470,169.704,33.823,156.385
C04697=1045.532,-48.727,-74.457,169.702,33.822,156.385
C04698=1045.526,-48.977,-74.444,169.700,33.821,156.385
C04699=1045.520,-49.227,-74.432,169.697,33.820,156.385
C04700=1045.513,-49.476,-74.420,169.695,33.819,156.385
C04701=1045.507,-49.726,-74.407,169.693,33.818,156.385
C04702=1045.501,-49.975,-74.394,169.691,33.817,156.385
C04703=1045.495,-50.225,-74.382,169.689,33.816,156.384
C04704=1045.488,-50.475,-74.370,169.687,33.815,156.384
C04705=1045.482,-50.724,-74.356,169.685,33.814,156.384
C04706=1045.474,-51.006,-74.343,169.682,33.813,156.384
C04707=1045.467,-51.287,-74.329,169.680,33.812,156.384
C04708=1045.460,-51.568,-74.315,169.679,33.812,156.384
C04709=1045.453,-51.849,-74.300,169.676,33.810,156.384
C04710=1045.446,-52.099,-74.288,169.674,33.809,156.384
C04711=1045.440,-52.349,-74.276,169.672,33.808,156.384
C04712=1045.434,-52.598,-74.264,169.670,33.808,156.384
C04713=1045.427,-52.848,-74.252,169.668,33.807,156.383
C04714=1045.421,-53.098,-74.239,169.666,33.806,156.383
C04715=1045.415,-53.348,-74.227,169.663,33.805,156.383
C04716=1045.408,-53.596,-74.215,169.661,33.804,156.383
C04717=1045.402,-53.846,-74.202,169.659,33.803,156.383
C04718=1045.395,-54.096,-74.190,169.657,33.802,156.383
C04719=1045.389,-54.346,-74.178,169.655,33.802,156.383
C04720=1045.383,-54.595,-74.166,169.653,33.801,156.383
C04721=1045.376,-54.845,-74.154,169.650,33.800,156.383
C04722=1045.371,-55.094,-74.142,169.648,33.799,156.383
C04723=1045.364,-55.344,-74.130,169.646,33.798,156.382
C04724=1045.358,-55.594,-74.117,169.644,33.797,156.382
C04725=1045.351,-55.843,-74.105,169.642,33.796,156.382
C04726=1045.345,-56.093,-74.093,169.640,33.795,156.382
C04727=1045.339,-56.343,-74.081,169.638,33.795,156.382
C04728=1045.332,-56.592,-74.069,169.635,33.794,156.382
C04729=1045.326,-56.842,-74.056,169.633,33.793,156.382
C04730=1045.320,-57.092,-74.044,169.631,33.792,156.382
C04731=1045.313,-57.341,-74.032,169.629,33.791,156.382
C04732=1045.307,-57.591,-74.020,169.627,33.790,156.382
C04733=1045.300,-57.841,-74.008,169.625,33.789,156.382
C04734=1045.294,-58.090,-73.996,169.622,33.788,156.382
C04735=1045.288,-58.339,-73.983,169.620,33.788,156.381
C04736=1045.282,-58.589,-73.971,169.618,33.787,156.381
C04737=1045.275,-58.839,-73.960,169.616,33.786,156.381
C04738=1045.269,-59.088,-73.947,169.614,33.785,156.381
C04739=1045.263,-59.338,-73.935,169.612,33.784,156.381
C04740=1045.256,-59.588,-73.923,169.609,33.784,156.381
C04741=1045.250,-59.837,-73.911,169.607,33.783,156.381
C04742=1045.244,-60.086,-73.899,169.605,33.781,156.381
C04743=1045.238,-60.336,-73.886,169.603,33.781,156.381
C04744=1045.232,-60.586,-73.875,169.601,33.780,156.381
C04745=1045.225,-60.836,-73.863,169.599,33.779,156.381
C04746=1045.219,-61.086,-73.851,169.596,33.778,156.380
C04747=1045.213,-61.335,-73.839,169.594,33.777,156.380
C04748=1045.206,-61.584,-73.827,169.592,33.777,156.380
C04749=1045.201,-61.834,-73.814,169.590,33.776,156.380
C04750=1045.194,-62.084,-73.803,169.588,33.775,156.380
C04751=1045.188,-62.334,-73.791,169.586,33.774,156.380
C04752=1045.182,-62.583,-73.780,169.583,33.773,156.380
C04753=1045.176,-62.833,-73.767,169.581,33.773,156.380
C04754=1045.169,-63.082,-73.755,169.579,33.772,156.380
C04755=1045.162,-63.332,-73.743,169.577,33.771,156.380
C04756=1045.157,-63.582,-73.731,169.575,33.770,156.380
C04757=1045.151,-63.831,-73.720,169.573,33.770,156.380
C04758=1045.144,-64.081,-73.708,169.570,33.769,156.380
C04759=1045.138,-64.331,-73.695,169.568,33.768,156.380
C04760=1045.132,-64.580,-73.683,169.566,33.767,156.379
C04761=1045.126,-64.830,-73.672,169.564,33.766,156.379
C04762=1045.120,-65.080,-73.660,169.562,33.766,156.379
C04763=1045.113,-65.329,-73.648,169.559,33.765,156.379
C04764=1045.107,-65.579,-73.637,169.557,33.764,156.379
C04765=1045.101,-65.828,-73.625,169.555,33.763,156.379
C04766=1045.095,-66.078,-73.613,169.553,33.762,156.379
C04767=1045.088,-66.328,-73.601,169.551,33.762,156.379
C04768=1045.083,-66.577,-73.590,169.548,33.761,156.379
C04769=1045.077,-66.827,-73.577,169.546,33.760,156.379
C04770=1045.070,-67.110,-73.564,169.544,33.759,156.379
C04771=1045.063,-67.392,-73.550,169.541,33.758,156.379
C04772=1045.056,-67.674,-73.537,169.539,33.757,156.378
C04773=1045.048,-67.957,-73.524,169.536,33.756,156.378
C04774=1045.043,-68.207,-73.512,169.534,33.755,156.378
C04775=1045.036,-68.456,-73.501,169.532,33.755,156.378
C04776=1045.030,-68.707,-73.489,169.530,33.754,156.378
C04777=1045.024,-68.956,-73.477,169.528,33.753,156.378
C04778=1045.018,-69.205,-73.465,169.525,33.752,156.378
C04779=1045.012,-69.455,-73.454,169.523,33.751,156.378
C04780=1045.005,-69.704,-73.442,169.521,33.751,156.378
C04781=1045.000,-69.955,-73.430,169.519,33.750,156.378
C04782=1044.994,-70.204,-73.419,169.517,33.749,156.378
C04783=1044.987,-70.453,-73.407,169.514,33.749,156.378
C04784=1044.981,-70.703,-73.396,169.512,33.748,156.378
C04785=1044.975,-70.953,-73.383,169.510,33.747,156.378
C04786=1044.969,-71.203,-73.372,169.508,33.746,156.378
C04787=1044.963,-71.452,-73.361,169.506,33.746,156.377
C04788=1044.957,-71.702,-73.349,169.503,33.745,156.377
C04789=1044.951,-71.952,-73.337,169.501,33.744,156.377
C04790=1044.945,-72.201,-73.326,169.499,33.743,156.377
C04791=1044.938,-72.451,-73.314,169.497,33.742,156.377
C04792=1044.933,-72.700,-73.303,169.495,33.742,156.377
C04793=1044.926,-72.950,-73.291,169.492,33.741,156.377
C04794=1044.921,-73.200,-73.280,169.490,33.740,156.377
C04795=1044.914,-73.449,-73.268,169.488,33.739,156.377
C04796=1044.909,-73.699,-73.257,169.486,33.739,156.377
C04797=1044.902,-73.948,-73.245,169.483,33.738,156.377
C04798=1044.896,-74.199,-73.234,169.481,33.737,156.377
C04799=1044.890,-74.448,-73.223,169.479,33.737,156.377
C04800=1044.883,-74.698,-73.211,169.477,33.736,156.377
C04801=1044.878,-74.947,-73.200,169.474,33.736,156.377
C04802=1044.871,-75.197,-73.188,169.472,33.735,156.377
C04803=1044.865,-75.447,-73.177,169.470,33.734,156.376
C04804=1044.859,-75.696,-73.166,169.468,33.734,156.377
C04805=1044.852,-75.946,-73.154,169.465,33.733,156.376
C04806=1044.846,-76.195,-73.143,169.463,33.732,156.376
C04807=1044.840,-76.446,-73.132,169.461,33.731,156.376
C04808=1044.834,-76.694,-73.120,169.459,33.731,156.376
C04809=1044.828,-76.945,-73.109,169.457,33.730,156.376
C04810=1044.822,-77.194,-73.098,169.455,33.730,156.376
C04811=1044.815,-77.444,-73.086,169.453,33.730,156.376
C04812=1044.810,-77.693,-73.075,169.451,33.729,156.376
C04813=1044.803,-77.943,-73.064,169.448,33.728,156.376
C04814=1044.797,-78.193,-73.053,169.446,33.728,156.376
C04815=1044.791,-78.442,-73.041,169.444,33.727,156.376
C04816=1044.785,-78.692,-73.030,169.442,33.726,156.376
C04817=1044.779,-78.942,-73.019,169.439,33.725,156.376
C04818=1044.773,-79.192,-73.008,169.437,33.725,156.376
C04819=1044.766,-79.441,-72.996,169.435,33.724,156.376
C04820=1044.760,-79.691,-72.985,169.433,33.724,156.376
C04821=1044.754,-79.941,-72.975,169.430,33.723,156.376
C04822=1044.747,-80.191,-72.963,169.428,33.723,156.376
C04823=1044.741,-80.440,-72.953,169.426,33.722,156.376
C04824=1044.735,-80.690,-72.941,169.424,33.722,156.376
C04825=1044.728,-80.939,-72.930,169.421,33.721,156.376
C04826=1044.722,-81.189,-72.919,169.419,33.721,156.376
C04827=1044.716,-81.439,-72.908,169.417,33.720,156.376
C04828=1044.709,-81.689,-72.898,169.414,33.720,156.376
C04829=1044.703,-81.938,-72.887,169.412,33.719,156.376
C04830=1044.697,-82.188,-72.875,169.410,33.719,156.376
C04831=1044.691,-82.438,-72.865,169.408,33.719,156.376
C04832=1044.684,-82.688,-72.854,169.405,33.718,156.376
C04833=1044.679,-82.937,-72.843,169.403,33.718,156.376
C04834=1044.671,-83.222,-72.830,169.400,33.717,156.376
C04835=1044.664,-83.506,-72.818,169.398,33.717,156.376
C04836=1044.657,-83.790,-72.805,169.395,33.716,156.376
C04837=1044.650,-84.076,-72.793,169.392,33.715,156.376
C04838=1044.644,-84.325,-72.782,169.390,33.715,156.376
C04839=1044.637,-84.575,-72.772,169.388,33.714,156.376
C04840=1044.631,-84.825,-72.761,169.386,33.714,156.376
C04841=1044.625,-85.075,-72.749,169.383,33.713,156.376
C04842=1044.618,-85.324,-72.739,169.381,33.713,156.376
C04843=1044.613,-85.574,-72.728,169.379,33.713,156.375
C04844=1044.606,-85.824,-72.717,169.376,33.712,156.376
C04845=1044.600,-86.073,-72.707,169.374,33.712,156.375
C04846=1044.594,-86.323,-72.696,169.372,33.711,156.375
C04847=1044.588,-86.573,-72.685,169.369,33.711,156.376
C04848=1044.581,-86.822,-72.674,169.367,33.710,156.375
C04849=1044.575,-87.072,-72.663,169.365,33.710,156.375
C04850=1044.569,-87.321,-72.652,169.363,33.709,156.375
C04851=1044.562,-87.571,-72.642,169.360,33.709,156.375
C04852=1044.556,-87.821,-72.631,169.358,33.709,156.375
C04853=1044.551,-88.070,-72.620,169.356,33.708,156.375
C04854=1044.544,-88.320,-72.609,169.353,33.708,156.375
C04855=1044.538,-88.570,-72.598,169.351,33.707,156.375
C04856=1044.532,-88.820,-72.588,169.349,33.707,156.375
C04857=1044.525,-89.070,-72.578,169.347,33.707,156.375
C04858=1044.520,-89.319,-72.567,169.345,33.706,156.375
C04859=1044.514,-89.569,-72.556,169.343,33.706,156.375
C04860=1044.507,-89.819,-72.545,169.340,33.705,156.375
C04861=1044.501,-90.068,-72.534,169.338,33.705,156.375
C04862=1044.495,-90.317,-72.524,169.336,33.705,156.375
C04863=1044.489,-90.568,-72.513,169.334,33.704,156.375
C04864=1044.483,-90.818,-72.503,169.331,33.704,156.375
C04865=1044.476,-91.067,-72.492,169.329,33.704,156.375
C04866=1044.471,-91.316,-72.481,169.327,33.703,156.375
C04867=1044.464,-91.566,-72.470,169.324,33.703,156.375
C04868=1044.458,-91.816,-72.461,169.322,33.702,156.375
C04869=1044.452,-92.066,-72.450,169.320,33.702,156.375
C04870=1044.446,-92.315,-72.439,169.317,33.701,156.375
C04871=1044.440,-92.565,-72.428,169.315,33.701,156.375
C04872=1044.434,-92.815,-72.417,169.313,33.701,156.375
C04873=1044.428,-93.064,-72.408,169.310,33.700,156.375
C04874=1044.422,-93.314,-72.397,169.308,33.700,156.375
C04875=1044.415,-93.564,-72.386,169.306,33.699,156.375
C04876=1044.409,-93.814,-72.376,169.303,33.699,156.375
C04877=1044.404,-94.063,-72.365,169.301,33.699,156.375
C04878=1044.397,-94.312,-72.355,169.299,33.699,156.376
C04879=1044.391,-94.563,-72.344,169.296,33.698,156.375
C04880=1044.385,-94.812,-72.334,169.294,33.698,156.376
C04881=1044.379,-95.062,-72.323,169.292,33.698,156.376
C04882=1044.373,-95.311,-72.312,169.289,33.697,156.375
C04883=1044.367,-95.561,-72.303,169.287,33.697,156.376
C04884=1044.361,-95.811,-72.292,169.285,33.696,156.376
C04885=1044.354,-96.061,-72.281,169.282,33.696,156.376
C04886=1044.349,-96.311,-72.271,169.280,33.695,156.376
C04887=1044.343,-96.560,-72.260,169.278,33.695,156.376
C04888=1044.337,-96.809,-72.250,169.275,33.695,156.376
C04889=1044.331,-97.059,-72.240,169.273,33.695,156.376
C04890=1044.324,-97.309,-72.229,169.271,33.694,156.376
C04891=1044.319,-97.559,-72.219,169.269,33.694,156.376
C04892=1044.312,-97.809,-72.209,169.266,33.694,156.376
C04893=1044.306,-98.058,-72.199,169.264,33.694,156.376
C04894=1044.300,-98.308,-72.188,169.261,33.693,156.376
C04895=1044.293,-98.558,-72.178,169.259,33.693,156.376
C04896=1044.288,-98.808,-72.167,169.257,33.693,156.376
C04897=1044.282,-99.058,-72.158,169.255,33.693,156.376
C04898=1044.273,-99.384,-72.144,169.252,33.693,156.376
C04899=1044.265,-99.710,-72.131,169.249,33.692,156.376
C04900=1044.258,-100.035,-72.117,169.246,33.692,156.376
C04901=1044.249,-100.361,-72.105,169.243,33.691,156.376
C04902=1044.243,-100.612,-72.095,169.241,33.691,156.376
C04903=1044.237,-100.861,-72.084,169.238,33.691,156.376
C04904=1044.230,-101.111,-72.074,169.236,33.691,156.376
C04905=1044.224,-101.361,-72.063,169.234,33.691,156.376
C04906=1044.218,-101.611,-72.054,169.231,33.690,156.376
C04907=1044.212,-101.860,-72.044,169.229,33.690,156.376
C04908=1044.206,-102.110,-72.033,169.226,33.690,156.376
C04909=1044.200,-102.360,-72.024,169.224,33.690,156.376
C04910=1044.194,-102.609,-72.014,169.222,33.690,156.376
C04911=1044.188,-102.859,-72.003,169.219,33.690,156.376
C04912=1044.182,-103.108,-71.993,169.217,33.689,156.376
C04913=1044.176,-103.358,-71.984,169.215,33.689,156.376
C04914=1044.169,-103.609,-71.973,169.212,33.689,156.376
C04915=1044.163,-103.858,-71.963,169.210,33.689,156.377
C04916=1044.157,-104.108,-71.953,169.208,33.689,156.377
C04917=1044.151,-104.357,-71.944,169.205,33.688,156.377
C04918=1044.145,-104.607,-71.933,169.203,33.688,156.377
C04919=1044.139,-104.857,-71.923,169.200,33.688,156.377
C04920=1044.133,-105.107,-71.914,169.198,33.688,156.377
C04921=1044.126,-105.356,-71.903,169.196,33.688,156.377
C04922=1044.121,-105.606,-71.893,169.193,33.688,156.377
C04923=1044.115,-105.856,-71.884,169.191,33.687,156.377
C04924=1044.108,-106.105,-71.874,169.189,33.688,156.377
C04925=1044.102,-106.355,-71.864,169.186,33.688,156.377
C04926=1044.096,-106.605,-71.854,169.184,33.688,156.377
C04927=1044.090,-106.855,-71.844,169.181,33.687,156.377
C04928=1044.084,-107.104,-71.835,169.179,33.687,156.377
C04929=1044.078,-107.353,-71.824,169.178,33.687,156.377
C04930=1044.071,-107.603,-71.815,169.175,33.687,156.377
C04931=1044.066,-107.853,-71.804,169.173,33.687,156.377
C04932=1044.060,-108.103,-71.795,169.170,33.687,156.377
C04933=1044.054,-108.353,-71.785,169.168,33.687,156.377
C04934=1044.047,-108.602,-71.775,169.166,33.687,156.378
C04935=1044.041,-108.852,-71.766,169.163,33.687,156.378
C04936=1044.035,-109.102,-71.756,169.161,33.686,156.378
C04937=1044.029,-109.352,-71.746,169.158,33.687,156.378
C04938=1044.022,-109.601,-71.737,169.156,33.687,156.378
C04939=1044.016,-109.851,-71.727,169.154,33.686,156.378
C04940=1044.010,-110.100,-71.717,169.151,33.686,156.378
C04941=1044.004,-110.350,-71.707,169.149,33.686,156.378
C04942=1043.998,-110.600,-71.697,169.146,33.687,156.378
C04943=1043.992,-110.850,-71.688,169.144,33.686,156.378
C04944=1043.986,-111.100,-71.678,169.142,33.686,156.378
C04945=1043.980,-111.350,-71.669,169.139,33.686,156.378
C04946=1043.974,-111.599,-71.659,169.137,33.686,156.378
C04947=1043.967,-111.849,-71.649,169.134,33.686,156.378
C04948=1043.961,-112.099,-71.640,169.132,33.686,156.378
C04949=1043.955,-112.349,-71.630,169.130,33.686,156.378
C04950=1043.949,-112.599,-71.621,169.127,33.686,156.379
C04951=1043.943,-112.848,-71.611,169.125,33.686,156.379
C04952=1043.937,-113.098,-71.602,169.122,33.686,156.379
C04953=1043.931,-113.347,-71.592,169.120,33.686,156.379
C04954=1043.925,-113.597,-71.583,169.118,33.686,156.379
C04955=1043.919,-113.847,-71.573,169.115,33.686,156.379
C04956=1043.913,-114.097,-71.563,169.113,33.686,156.379
C04957=1043.907,-114.347,-71.553,169.110,33.686,156.379
C04958=1043.896,-114.767,-71.537,169.107,33.686,156.379
C04959=1043.886,-115.189,-71.522,169.103,33.686,156.379
C04960=1043.879,-115.475,-71.511,169.100,33.687,156.380
C04961=1043.872,-115.761,-71.500,169.098,33.687,156.380
C04962=1043.865,-116.047,-71.489,169.095,33.686,156.380
C04963=1043.857,-116.333,-71.478,169.092,33.687,156.380
C04964=1043.852,-116.582,-71.469,169.090,33.687,156.380
C04965=1043.846,-116.832,-71.460,169.087,33.687,156.380
C04966=1043.840,-117.082,-71.451,169.085,33.687,156.380
C04967=1043.833,-117.332,-71.441,169.082,33.687,156.380
C04968=1043.827,-117.582,-71.431,169.080,33.687,156.380
C04969=1043.821,-117.832,-71.422,169.078,33.687,156.380
C04970=1043.815,-118.081,-71.413,169.075,33.687,156.380
C04971=1043.809,-118.330,-71.403,169.073,33.687,156.380
C04972=1043.803,-118.581,-71.394,169.070,33.688,156.381
C04973=1043.797,-118.831,-71.385,169.068,33.688,156.381
C04974=1043.790,-119.080,-71.376,169.065,33.688,156.381
C04975=1043.784,-119.330,-71.366,169.063,33.688,156.381
C04976=1043.779,-119.579,-71.357,169.061,33.688,156.381
C04977=1043.773,-119.829,-71.348,169.058,33.688,156.381
C04978=1043.767,-120.079,-71.339,169.056,33.689,156.381
C04979=1043.760,-120.329,-71.329,169.053,33.688,156.381
C04980=1043.754,-120.579,-71.319,169.051,33.689,156.381
C04981=1043.749,-120.828,-71.310,169.048,33.689,156.381
C04982=1043.742,-121.078,-71.302,169.046,33.689,156.382
C04983=1043.736,-121.328,-71.292,169.044,33.689,156.382
C04984=1043.730,-121.578,-71.283,169.042,33.689,156.382
C04985=1043.724,-121.827,-71.274,169.040,33.689,156.382
C04986=1043.718,-122.077,-71.265,169.037,33.690,156.382
C04987=1043.711,-122.327,-71.256,169.035,33.690,156.382
C04988=1043.705,-122.576,-71.246,169.032,33.690,156.382
C04989=1043.700,-122.826,-71.238,169.030,33.690,156.382
C04990=1043.694,-123.076,-71.228,169.028,33.690,156.382
C04991=1043.688,-123.326,-71.219,169.025,33.691,156.383
C04992=1043.682,-123.576,-71.210,169.023,33.691,156.383
C04993=1043.675,-123.825,-71.201,169.020,33.691,156.383
C04994=1043.669,-124.075,-71.192,169.018,33.691,156.383
C04995=1043.663,-124.325,-71.183,169.015,33.691,156.383
C04996=1043.657,-124.575,-71.173,169.013,33.692,156.383
C04997=1043.651,-124.824,-71.165,169.010,33.692,156.383
C04998=1043.645,-125.074,-71.156,169.008,33.692,156.383
C04999=1043.639,-125.324,-71.146,169.006,33.693,156.383
C05000=1043.633,-125.573,-71.138,169.003,33.693,156.384
C05001=1043.627,-125.823,-71.129,169.001,33.693,156.384
C05002=1043.621,-126.074,-71.120,168.998,33.693,156.384
C05003=1043.615,-126.322,-71.111,168.996,33.694,156.384
C05004=1043.609,-126.573,-71.102,168.993,33.693,156.384
C05005=1043.602,-126.823,-71.093,168.991,33.694,156.384
C05006=1043.596,-127.073,-71.085,168.988,33.694,156.384
C05007=1043.590,-127.322,-71.075,168.986,33.695,156.384
C05008=1043.584,-127.572,-71.066,168.983,33.695,156.384
C05009=1043.578,-127.821,-71.058,168.981,33.695,156.385
C05010=1043.573,-128.071,-71.048,168.980,33.695,156.385
C05011=1043.569,-128.321,-71.037,168.977,33.694,156.385
C05012=1043.565,-128.571,-71.027,168.975,33.693,156.385
C05013=1043.562,-128.820,-71.016,168.973,33.692,156.384
C05014=1043.561,-129.070,-71.004,168.972,33.690,156.384
C05015=1043.560,-129.320,-70.992,168.970,33.688,156.384
C05016=1043.560,-129.571,-70.979,168.967,33.684,156.383
C05017=1043.561,-129.821,-70.965,168.966,33.681,156.383
C05018=1043.563,-130.071,-70.950,168.964,33.678,156.382
C05019=1043.565,-130.321,-70.935,168.963,33.673,156.381
C05020=1043.569,-130.572,-70.919,168.962,33.669,156.381
C05021=1043.573,-130.822,-70.903,168.961,33.663,156.380
C05022=1043.579,-131.073,-70.887,168.960,33.658,156.379
C05023=1043.584,-131.322,-70.870,168.960,33.652,156.378
C05024=1043.233,-131.346,-71.117,168.913,33.837,156.411
C05025=1043.226,-131.096,-71.135,168.914,33.843,156.412
C05026=1043.220,-130.846,-71.152,168.915,33.849,156.413
C05027=1043.216,-130.595,-71.168,168.916,33.854,156.414
C05028=1043.213,-130.345,-71.184,168.917,33.859,156.414
C05029=1043.209,-130.095,-71.198,168.918,33.863,156.415
C05030=1043.208,-129.845,-71.213,168.919,33.867,156.416
C05031=1043.208,-129.595,-71.227,168.922,33.870,156.416
C05032=1043.207,-129.345,-71.240,168.923,33.873,156.417
C05033=1043.208,-129.094,-71.252,168.925,33.875,156.417
C05034=1043.209,-128.844,-71.264,168.927,33.877,156.417
C05035=1043.212,-128.595,-71.276,168.929,33.879,156.417
C05036=1043.216,-128.344,-71.286,168.931,33.880,156.417
C05037=1043.220,-128.095,-71.296,168.933,33.880,156.418
C05038=1043.225,-127.845,-71.306,168.935,33.881,156.418
C05039=1043.232,-127.596,-71.315,168.938,33.880,156.417
C05040=1043.237,-127.346,-71.323,168.940,33.880,156.417
C05041=1043.243,-127.096,-71.333,168.942,33.880,156.417
C05042=1043.250,-126.846,-71.341,168.944,33.879,156.417
C05043=1043.255,-126.597,-71.350,168.947,33.879,156.417
C05044=1043.261,-126.347,-71.359,168.949,33.879,156.417
C05045=1043.268,-126.097,-71.368,168.952,33.879,156.417
C05046=1043.273,-125.847,-71.377,168.954,33.878,156.417
C05047=1043.280,-125.598,-71.386,168.957,33.878,156.416
C05048=1043.287,-125.348,-71.395,168.959,33.878,156.416
C05049=1043.292,-125.098,-71.404,168.961,33.877,156.416
C05050=1043.298,-124.849,-71.413,168.964,33.877,156.416
C05051=1043.305,-124.599,-71.422,168.966,33.876,156.416
C05052=1043.311,-124.349,-71.431,168.969,33.877,156.416
C05053=1043.316,-124.099,-71.440,168.971,33.876,156.416
C05054=1043.322,-123.849,-71.449,168.974,33.876,156.416
C05055=1043.328,-123.599,-71.459,168.976,33.876,156.416
C05056=1043.335,-123.349,-71.467,168.979,33.875,156.415
C05057=1043.341,-123.100,-71.476,168.981,33.875,156.415
C05058=1043.347,-122.850,-71.486,168.984,33.875,156.415
C05059=1043.353,-122.600,-71.495,168.986,33.875,156.415
C05060=1043.358,-122.351,-71.504,168.988,33.875,156.415
C05061=1043.365,-122.101,-71.513,168.991,33.874,156.415
C05062=1043.371,-121.851,-71.522,168.993,33.874,156.415
C05063=1043.377,-121.601,-71.531,168.996,33.874,156.415
C05064=1043.383,-121.351,-71.541,168.998,33.874,156.415
C05065=1043.389,-121.102,-71.550,169.001,33.874,156.414
C05066=1043.395,-120.852,-71.559,169.002,33.873,156.414
C05067=1043.402,-120.602,-71.568,169.005,33.873,156.414
C05068=1043.408,-120.353,-71.577,169.007,33.873,156.414
C05069=1043.413,-120.104,-71.587,169.010,33.873,156.414
C05070=1043.419,-119.853,-71.595,169.012,33.873,156.414
C05071=1043.425,-119.603,-71.605,169.014,33.873,156.414
C05072=1043.432,-119.354,-71.615,169.017,33.872,156.414
C05073=1043.438,-119.104,-71.624,169.019,33.872,156.414
C05074=1043.444,-118.855,-71.633,169.022,33.872,156.414
C05075=1043.450,-118.605,-71.642,169.024,33.872,156.414
C05076=1043.456,-118.355,-71.651,169.027,33.872,156.413
C05077=1043.462,-118.105,-71.661,169.029,33.872,156.413
C05078=1043.468,-117.855,-71.670,169.031,33.871,156.413
C05079=1043.475,-117.605,-71.680,169.034,33.872,156.413
C05080=1043.480,-117.356,-71.689,169.036,33.871,156.413
C05081=1043.486,-117.106,-71.698,169.039,33.871,156.413
C05082=1043.492,-116.856,-71.707,169.041,33.871,156.413
C05083=1043.498,-116.606,-71.717,169.044,33.871,156.413
C05084=1043.505,-116.356,-71.727,169.046,33.870,156.413
C05085=1043.512,-116.070,-71.737,169.049,33.871,156.413
C05086=1043.518,-115.785,-71.748,169.052,33.870,156.412
C05087=1043.526,-115.499,-71.758,169.054,33.870,156.412
C05088=1043.533,-115.213,-71.770,169.057,33.870,156.412
C05089=1043.539,-114.963,-71.780,169.060,33.870,156.412
C05090=1043.545,-114.714,-71.789,169.062,33.870,156.412
C05091=1043.551,-114.464,-71.798,169.065,33.870,156.412
C05092=1043.557,-114.213,-71.807,169.067,33.870,156.412
C05093=1043.563,-113.964,-71.817,169.069,33.870,156.412
C05094=1043.569,-113.714,-71.826,169.071,33.870,156.412
C05095=1043.575,-113.464,-71.836,169.073,33.870,156.412
C05096=1043.581,-113.214,-71.845,169.076,33.870,156.412
C05097=1043.587,-112.965,-71.855,169.078,33.870,156.412
C05098=1043.594,-112.715,-71.865,169.080,33.870,156.411
C05099=1043.600,-112.466,-71.875,169.083,33.870,156.411
C05100=1043.606,-112.216,-71.884,169.085,33.869,156.411
C05101=1043.612,-111.967,-71.894,169.088,33.870,156.411
C05102=1043.618,-111.717,-71.903,169.090,33.870,156.411
C05103=1043.624,-111.467,-71.913,169.093,33.869,156.411
C05104=1043.630,-111.217,-71.922,169.095,33.869,156.411
C05105=1043.637,-110.967,-71.932,169.097,33.870,156.411
C05106=1043.642,-110.717,-71.942,169.100,33.870,156.411
C05107=1043.648,-110.468,-71.952,169.102,33.869,156.411
C05108=1043.654,-110.218,-71.961,169.105,33.870,156.411
C05109=1043.661,-109.968,-71.971,169.107,33.870,156.411
C05110=1043.667,-109.718,-71.980,169.109,33.870,156.411
C05111=1043.673,-109.469,-71.991,169.112,33.869,156.411
C05112=1043.679,-109.219,-72.000,169.114,33.870,156.410
C05113=1043.686,-108.969,-72.010,169.117,33.870,156.410
C05114=1043.692,-108.720,-72.019,169.119,33.870,156.410
C05115=1043.698,-108.470,-72.029,169.122,33.869,156.410
C05116=1043.704,-108.220,-72.038,169.124,33.870,156.410
C05117=1043.710,-107.970,-72.049,169.126,33.870,156.410
C05118=1043.716,-107.721,-72.059,169.129,33.870,156.410
C05119=1043.722,-107.471,-72.068,169.131,33.869,156.410
C05120=1043.728,-107.221,-72.078,169.134,33.870,156.410
C05121=1043.734,-106.971,-72.088,169.136,33.870,156.410
C05122=1043.741,-106.722,-72.098,169.138,33.870,156.410
C05123=1043.746,-106.472,-72.108,169.141,33.870,156.410
C05124=1043.753,-106.222,-72.118,169.142,33.870,156.410
C05125=1043.759,-105.972,-72.127,169.144,33.870,156.410
C05126=1043.765,-105.723,-72.137,169.147,33.870,156.410
C05127=1043.771,-105.473,-72.148,169.149,33.870,156.410
C05128=1043.777,-105.223,-72.157,169.152,33.870,156.410
C05129=1043.783,-104.974,-72.167,169.154,33.870,156.409
C05130=1043.789,-104.724,-72.177,169.156,33.871,156.409
C05131=1043.795,-104.474,-72.187,169.159,33.871,156.409
C05132=1043.801,-104.225,-72.197,169.161,33.871,156.409
C05133=1043.808,-103.975,-72.207,169.164,33.871,156.409
C05134=1043.814,-103.725,-72.217,169.166,33.871,156.409
C05135=1043.820,-103.475,-72.228,169.168,33.871,156.409
C05136=1043.826,-103.225,-72.237,169.171,33.872,156.409
C05137=1043.832,-102.976,-72.247,169.173,33.872,156.409
C05138=1043.838,-102.726,-72.258,169.176,33.872,156.409
C05139=1043.844,-102.476,-72.267,169.178,33.872,156.409
C05140=1043.850,-102.227,-72.277,169.180,33.872,156.409
C05141=1043.856,-101.977,-72.288,169.183,33.873,156.409
C05142=1043.862,-101.727,-72.297,169.185,33.873,156.409
C05143=1043.869,-101.478,-72.308,169.187,33.873,156.409
C05144=1043.875,-101.227,-72.318,169.190,33.873,156.409
C05145=1043.881,-100.978,-72.329,169.192,33.873,156.409
C05146=1043.888,-100.728,-72.338,169.195,33.873,156.409
C05147=1043.894,-100.479,-72.348,169.197,33.874,156.409
C05148=1043.899,-100.229,-72.359,169.199,33.874,156.409
C05149=1043.907,-99.942,-72.370,169.202,33.874,156.409
C05150=1043.914,-99.655,-72.382,169.205,33.874,156.409
C05151=1043.921,-99.367,-72.394,169.207,33.874,156.409
C05152=1043.928,-99.081,-72.405,169.210,33.874,156.409
C05153=1043.934,-98.832,-72.415,169.213,33.875,156.409
C05154=1043.940,-98.581,-72.426,169.215,33.875,156.409
C05155=1043.947,-98.332,-72.436,169.217,33.875,156.408
C05156=1043.953,-98.082,-72.446,169.220,33.875,156.408
C05157=1043.959,-97.832,-72.456,169.222,33.875,156.408
C05158=1043.965,-97.583,-72.466,169.224,33.875,156.408
C05159=1043.971,-97.333,-72.477,169.226,33.876,156.408
C05160=1043.978,-97.083,-72.487,169.228,33.876,156.408
C05161=1043.983,-96.834,-72.498,169.230,33.877,156.408
C05162=1043.989,-96.584,-72.507,169.233,33.877,156.408
C05163=1043.995,-96.334,-72.518,169.235,33.877,156.408
C05164=1044.001,-96.085,-72.529,169.237,33.877,156.408
C05165=1044.012,-95.675,-72.546,169.241,33.878,156.408
C05166=1044.022,-95.267,-72.563,169.245,33.878,156.408
C05167=1044.031,-94.858,-72.580,169.249,33.879,156.408
C05168=1044.041,-94.450,-72.597,169.253,33.879,156.408
C05169=1044.047,-94.200,-72.608,169.255,33.880,156.408
C05170=1044.054,-93.950,-72.618,169.257,33.880,156.408
C05171=1044.059,-93.700,-72.629,169.260,33.881,156.408
C05172=1044.065,-93.451,-72.640,169.262,33.881,156.408
C05173=1044.071,-93.201,-72.649,169.264,33.881,156.408
C05174=1044.077,-92.951,-72.660,169.267,33.881,156.408
C05175=1044.084,-92.702,-72.671,169.269,33.882,156.408
C05176=1044.090,-92.452,-72.682,169.271,33.882,156.408
C05177=1044.095,-92.202,-72.692,169.274,33.882,156.408
C05178=1044.102,-91.953,-72.702,169.276,33.883,156.408
C05179=1044.108,-91.703,-72.714,169.278,33.883,156.408
C05180=1044.115,-91.453,-72.724,169.281,33.883,156.408
C05181=1044.120,-91.204,-72.735,169.283,33.883,156.408
C05182=1044.126,-90.953,-72.745,169.285,33.884,156.408
C05183=1044.133,-90.704,-72.756,169.288,33.884,156.408
C05184=1044.139,-90.454,-72.766,169.290,33.885,156.408
C05185=1044.144,-90.205,-72.777,169.292,33.885,156.408
C05186=1044.151,-89.955,-72.788,169.295,33.886,156.408
C05187=1044.157,-89.706,-72.799,169.297,33.886,156.408
C05188=1044.163,-89.455,-72.809,169.299,33.886,156.408
C05189=1044.170,-89.206,-72.820,169.302,33.887,156.408
C05190=1044.175,-88.956,-72.830,169.304,33.887,156.408
C05191=1044.182,-88.707,-72.841,169.306,33.888,156.408
C05192=1044.188,-88.457,-72.852,169.309,33.888,156.408
C05193=1044.194,-88.207,-72.863,169.311,33.888,156.408
C05194=1044.201,-87.958,-72.873,169.313,33.889,156.408
C05195=1044.207,-87.708,-72.884,169.316,33.889,156.408
C05196=1044.213,-87.458,-72.895,169.318,33.889,156.408
C05197=1044.219,-87.208,-72.905,169.320,33.890,156.408
C05198=1044.225,-86.958,-72.916,169.323,33.890,156.408
C05199=1044.231,-86.709,-72.927,169.325,33.891,156.408
C05200=1044.238,-86.459,-72.938,169.327,33.891,156.408
C05201=1044.244,-86.209,-72.948,169.329,33.891,156.408
C05202=1044.249,-85.960,-72.959,169.332,33.892,156.408
C05203=1044.256,-85.710,-72.970,169.334,33.892,156.408
C05204=1044.262,-85.461,-72.981,169.335,33.892,156.408
C05205=1044.269,-85.210,-72.992,169.338,33.893,156.408
C05206=1044.275,-84.961,-73.002,169.340,33.893,156.408
C05207=1044.281,-84.711,-73.014,169.342,33.894,156.408
C05208=1044.287,-84.462,-73.025,169.345,33.894,156.408
C05209=1044.297,-84.086,-73.041,169.348,33.895,156.408
C05210=1044.307,-83.711,-73.057,169.352,33.895,156.408
C05211=1044.315,-83.336,-73.073,169.355,33.896,156.408
C05212=1044.325,-82.961,-73.090,169.359,33.897,156.408
C05213=1044.331,-82.711,-73.102,169.361,33.897,156.408
C05214=1044.338,-82.461,-73.112,169.363,33.897,156.408
C05215=1044.344,-82.211,-73.123,169.365,33.898,156.408
C05216=1044.350,-81.962,-73.134,169.368,33.898,156.408
C05217=1044.356,-81.712,-73.145,169.370,33.899,156.408
C05218=1044.363,-81.462,-73.156,169.372,33.899,156.408
C05219=1044.369,-81.212,-73.167,169.375,33.900,156.408
C05220=1044.375,-80.963,-73.178,169.377,33.900,156.408
C05221=1044.382,-80.713,-73.189,169.379,33.901,156.408
C05222=1044.388,-80.464,-73.200,169.382,33.901,156.408
C05223=1044.394,-80.214,-73.211,169.384,33.902,156.408
C05224=1044.400,-79.964,-73.222,169.386,33.902,156.408
C05225=1044.407,-79.714,-73.233,169.388,33.903,156.408
C05226=1044.413,-79.465,-73.244,169.391,33.903,156.408
C05227=1044.419,-79.215,-73.255,169.393,33.904,156.409
C05228=1044.425,-78.966,-73.266,169.395,33.904,156.408
C05229=1044.432,-78.716,-73.278,169.397,33.905,156.409
C05230=1044.437,-78.466,-73.288,169.400,33.906,156.409
C05231=1044.444,-78.217,-73.300,169.402,33.906,156.409
C05232=1044.450,-77.967,-73.311,169.404,33.907,156.409
C05233=1044.456,-77.717,-73.323,169.407,33.908,156.409
C05234=1044.462,-77.467,-73.333,169.409,33.908,156.409
C05235=1044.468,-77.218,-73.345,169.411,33.908,156.409
C05236=1044.474,-76.968,-73.356,169.413,33.909,156.409
C05237=1044.480,-76.718,-73.368,169.416,33.909,156.409
C05238=1044.487,-76.469,-73.379,169.418,33.910,156.409
C05239=1044.493,-76.219,-73.390,169.420,33.911,156.409
C05240=1044.499,-75.970,-73.401,169.422,33.911,156.409
C05241=1044.505,-75.720,-73.413,169.425,33.912,156.409
C05242=1044.512,-75.470,-73.424,169.427,33.913,156.409
C05243=1044.517,-75.220,-73.435,169.429,33.913,156.409
C05244=1044.524,-74.971,-73.447,169.431,33.914,156.409
C05245=1044.530,-74.721,-73.458,169.434,33.914,156.409
C05246=1044.536,-74.471,-73.469,169.436,33.915,156.409
C05247=1044.543,-74.222,-73.481,169.438,33.915,156.409
C05248=1044.548,-73.972,-73.492,169.440,33.916,156.409
C05249=1044.555,-73.722,-73.504,169.443,33.917,156.409
C05250=1044.561,-73.473,-73.515,169.445,33.917,156.409
C05251=1044.567,-73.223,-73.527,169.447,33.918,156.409
C05252=1044.573,-72.974,-73.538,169.449,33.919,156.410
C05253=1044.579,-72.724,-73.550,169.451,33.919,156.410
C05254=1044.585,-72.475,-73.561,169.454,33.920,156.410
C05255=1044.591,-72.225,-73.573,169.456,33.921,156.410
C05256=1044.598,-71.975,-73.585,169.458,33.922,156.410
C05257=1044.603,-71.726,-73.597,169.460,33.923,156.410
C05258=1044.609,-71.475,-73.608,169.463,33.923,156.410
C05259=1044.616,-71.227,-73.620,169.465,33.924,156.410
C05260=1044.622,-70.976,-73.631,169.467,33.924,156.410
C05261=1044.629,-70.727,-73.643,169.469,33.925,156.410
C05262=1044.634,-70.477,-73.654,169.471,33.926,156.410
C05263=1044.640,-70.227,-73.666,169.474,33.927,156.410
C05264=1044.646,-69.978,-73.677,169.476,33.928,156.410
C05265=1044.653,-69.728,-73.689,169.478,33.928,156.410
C05266=1044.658,-69.478,-73.702,169.480,33.929,156.410
C05267=1044.664,-69.229,-73.712,169.482,33.930,156.411
C05268=1044.671,-68.979,-73.724,169.485,33.931,156.411
C05269=1044.676,-68.729,-73.736,169.487,33.931,156.411
C05270=1044.682,-68.480,-73.748,169.489,33.932,156.411
C05271=1044.689,-68.230,-73.760,169.491,33.932,156.411
C05272=1044.695,-67.980,-73.771,169.494,33.933,156.411
C05273=1044.703,-67.698,-73.785,169.496,33.934,156.411
C05274=1044.709,-67.416,-73.798,169.499,33.935,156.411
C05275=1044.716,-67.133,-73.811,169.501,33.936,156.411
C05276=1044.723,-66.851,-73.824,169.503,33.937,156.411
C05277=1044.729,-66.600,-73.836,169.506,33.937,156.411
C05278=1044.735,-66.351,-73.848,169.508,33.938,156.411
C05279=1044.741,-66.102,-73.860,169.510,33.939,156.411
C05280=1044.748,-65.852,-73.872,169.512,33.940,156.411
C05281=1044.754,-65.602,-73.884,169.514,33.940,156.411
C05282=1044.760,-65.353,-73.895,169.516,33.941,156.412
C05283=1044.766,-65.103,-73.907,169.518,33.942,156.412
C05284=1044.772,-64.853,-73.919,169.520,33.943,156.412
C05285=1044.779,-64.603,-73.931,169.522,33.944,156.412
C05286=1044.785,-64.354,-73.943,169.524,33.944,156.412
C05287=1044.791,-64.105,-73.955,169.527,33.945,156.412
C05288=1044.797,-63.855,-73.967,169.529,33.946,156.412
C05289=1044.803,-63.605,-73.978,169.531,33.947,156.412
C05290=1044.810,-63.356,-73.990,169.533,33.947,156.412
C05291=1044.815,-63.106,-74.003,169.535,33.948,156.412
C05292=1044.822,-62.856,-74.014,169.538,33.949,156.412
C05293=1044.829,-62.607,-74.026,169.540,33.950,156.412
C05294=1044.834,-62.356,-74.038,169.542,33.951,156.412
C05295=1044.840,-62.107,-74.050,169.544,33.951,156.413
C05296=1044.847,-61.858,-74.062,169.546,33.952,156.413
C05297=1044.853,-61.608,-74.074,169.549,33.953,156.413
C05298=1044.860,-61.358,-74.086,169.551,33.954,156.413
C05299=1044.866,-61.109,-74.098,169.553,33.955,156.413
C05300=1044.871,-60.859,-74.110,169.555,33.955,156.413
C05301=1044.878,-60.609,-74.122,169.557,33.956,156.413
C05302=1044.885,-60.360,-74.134,169.559,33.957,156.413
C05303=1044.890,-60.110,-74.146,169.562,33.958,156.413
C05304=1044.897,-59.860,-74.158,169.564,33.958,156.413
C05305=1044.904,-59.611,-74.170,169.566,33.959,156.413
C05306=1044.909,-59.362,-74.182,169.568,33.960,156.413
C05307=1044.916,-59.112,-74.194,169.570,33.961,156.414
C05308=1044.922,-58.863,-74.206,169.572,33.962,156.414
C05309=1044.928,-58.613,-74.219,169.575,33.962,156.414
C05310=1044.935,-58.363,-74.231,169.577,33.963,156.414
C05311=1044.942,-58.114,-74.243,169.579,33.964,156.414
C05312=1044.947,-57.864,-74.255,169.581,33.965,156.414
C05313=1044.954,-57.613,-74.267,169.583,33.966,156.414
C05314=1044.959,-57.364,-74.279,169.585,33.967,156.414
C05315=1044.966,-57.115,-74.291,169.588,33.968,156.414
C05316=1044.972,-56.865,-74.303,169.590,33.968,156.414
C05317=1044.978,-56.615,-74.315,169.592,33.969,156.414
C05318=1044.985,-56.366,-74.327,169.594,33.970,156.414
C05319=1044.992,-56.117,-74.340,169.596,33.971,156.415
C05320=1044.998,-55.867,-74.352,169.598,33.972,156.415
C05321=1045.004,-55.617,-74.364,169.601,33.972,156.415
C05322=1045.010,-55.367,-74.377,169.603,33.973,156.415
C05323=1045.017,-55.118,-74.389,169.605,33.974,156.415
C05324=1045.024,-54.868,-74.401,169.607,33.975,156.415
C05325=1045.030,-54.618,-74.413,169.609,33.975,156.415
C05326=1045.036,-54.369,-74.425,169.611,33.976,156.415
C05327=1045.043,-54.119,-74.437,169.614,33.978,156.415
C05328=1045.049,-53.869,-74.450,169.616,33.978,156.415
C05329=1045.055,-53.620,-74.462,169.618,33.979,156.415
C05330=1045.061,-53.370,-74.474,169.620,33.980,156.416
C05331=1045.068,-53.120,-74.486,169.622,33.981,156.416
C05332=1045.075,-52.871,-74.499,169.624,33.982,156.416
C05333=1045.081,-52.621,-74.512,169.626,33.982,156.416
C05334=1045.087,-52.372,-74.523,169.629,33.983,156.416
C05335=1045.093,-52.122,-74.536,169.631,33.984,156.416
C05336=1045.100,-51.872,-74.548,169.633,33.985,156.416
C05337=1045.107,-51.592,-74.562,169.635,33.986,156.416
C05338=1045.114,-51.310,-74.576,169.638,33.987,156.416
C05339=1045.121,-51.029,-74.589,169.640,33.988,156.416
C05340=1045.129,-50.748,-74.604,169.643,33.989,156.417
C05341=1045.135,-50.498,-74.616,169.645,33.990,156.417
C05342=1045.141,-50.248,-74.628,169.647,33.991,156.417
C05343=1045.147,-49.999,-74.641,169.649,33.991,156.417
C05344=1045.153,-49.749,-74.654,169.651,33.993,156.417
C05345=1045.160,-49.500,-74.666,169.653,33.994,156.417
C05346=1045.166,-49.250,-74.679,169.655,33.994,156.417
C05347=1045.172,-49.001,-74.692,169.657,33.996,156.417
C05348=1045.178,-48.751,-74.704,169.659,33.997,156.417
C05349=1045.185,-48.501,-74.716,169.662,33.997,156.417
C05350=1045.191,-48.252,-74.730,169.664,33.999,156.418
C05351=1045.197,-48.002,-74.742,169.666,34.000,156.418
C05352=1045.203,-47.753,-74.755,169.668,34.000,156.418
C05353=1045.210,-47.503,-74.767,169.670,34.002,156.418
C05354=1045.216,-47.253,-74.780,169.672,34.002,156.418
C05355=1045.222,-47.004,-74.793,169.674,34.004,156.418
C05356=1045.228,-46.754,-74.806,169.676,34.005,156.418
C05357=1045.234,-46.504,-74.818,169.678,34.005,156.418
C05358=1045.241,-46.255,-74.831,169.680,34.007,156.419
C05359=1045.246,-46.005,-74.844,169.683,34.008,156.419
C05360=1045.253,-45.756,-74.857,169.685,34.008,156.419
C05361=1045.259,-45.506,-74.869,169.687,34.010,156.419
C05362=1045.265,-45.257,-74.881,169.689,34.011,156.419
C05363=1045.272,-45.007,-74.895,169.691,34.012,156.419
C05364=1045.278,-44.757,-74.907,169.693,34.013,156.419
C05365=1045.284,-44.508,-74.921,169.695,34.014,156.419
C05366=1045.290,-44.258,-74.933,169.697,34.015,156.420
C05367=1045.297,-44.009,-74.946,169.699,34.016,156.420
C05368=1045.303,-43.759,-74.959,169.701,34.017,156.420
C05369=1045.309,-43.510,-74.972,169.703,34.018,156.420
C05370=1045.315,-43.260,-74.984,169.705,34.019,156.420
C05371=1045.322,-43.011,-74.997,169.709,34.020,156.420
C05372=1045.328,-42.761,-75.010,169.711,34.021,156.420
C05373=1045.335,-42.511,-75.023,169.713,34.022,156.421
C05374=1045.341,-42.261,-75.036,169.715,34.023,156.421
C05375=1045.347,-42.012,-75.049,169.717,34.024,156.421
C05376=1045.354,-41.762,-75.061,169.719,34.025,156.421
C05377=1045.360,-41.513,-75.074,169.721,34.026,156.421
C05378=1045.366,-41.263,-75.087,169.723,34.027,156.421
C05379=1045.372,-41.014,-75.100,169.725,34.028,156.421
C05380=1045.379,-40.764,-75.114,169.727,34.029,156.421
C05381=1045.385,-40.514,-75.126,169.729,34.030,156.422
C05382=1045.392,-40.265,-75.139,169.731,34.031,156.422
C05383=1045.397,-40.015,-75.152,169.733,34.032,156.422
C05384=1045.404,-39.766,-75.165,169.735,34.033,156.422
C05385=1045.410,-39.516,-75.178,169.737,34.035,156.422
C05386=1045.416,-39.266,-75.191,169.740,34.035,156.422
C05387=1045.423,-39.017,-75.204,169.742,34.036,156.422
C05388=1045.429,-38.767,-75.216,169.744,34.038,156.422
C05389=1045.435,-38.518,-75.229,169.746,34.038,156.423
C05390=1045.442,-38.269,-75.243,169.748,34.040,156.423
C05391=1045.448,-38.019,-75.256,169.750,34.041,156.423
C05392=1045.454,-37.768,-75.270,169.752,34.042,156.423
C05393=1045.460,-37.519,-75.283,169.754,34.043,156.423
C05394=1045.466,-37.270,-75.296,169.756,34.044,156.423
C05395=1045.472,-37.020,-75.309,169.758,34.045,156.423
C05396=1045.479,-36.770,-75.322,169.760,34.046,156.424
C05397=1045.485,-36.521,-75.336,169.762,34.048,156.424
C05398=1045.491,-36.272,-75.349,169.764,34.049,156.424
C05399=1045.497,-36.022,-75.361,169.766,34.050,156.424
C05400=1045.503,-35.772,-75.375,169.768,34.051,156.424
C05401=1045.511,-35.492,-75.390,169.770,34.053,156.424
C05402=1045.517,-35.211,-75.404,169.773,34.053,156.424
C05403=1045.525,-34.930,-75.420,169.775,34.055,156.425
C05404=1045.532,-34.650,-75.434,169.777,34.056,156.425
C05405=1045.539,-34.400,-75.448,169.779,34.058,156.425
C05406=1045.544,-34.150,-75.461,169.781,34.058,156.425
C05407=1045.550,-33.900,-75.474,169.783,34.060,156.425
C05408=1045.556,-33.651,-75.488,169.785,34.060,156.425
C05409=1045.563,-33.401,-75.501,169.787,34.062,156.426
C05410=1045.569,-33.152,-75.515,169.789,34.063,156.426
C05411=1045.575,-32.902,-75.528,169.791,34.064,156.426
C05412=1045.581,-32.653,-75.540,169.793,34.065,156.426
C05413=1045.588,-32.403,-75.554,169.795,34.066,156.426
C05414=1045.594,-32.153,-75.567,169.797,34.068,156.426
C05415=1045.601,-31.904,-75.581,169.799,34.069,156.427
C05416=1045.607,-31.654,-75.594,169.801,34.070,156.427
C05417=1045.614,-31.405,-75.607,169.803,34.071,156.427
C05418=1045.619,-31.155,-75.621,169.805,34.072,156.427
C05419=1045.626,-30.905,-75.635,169.807,34.073,156.427
C05420=1045.632,-30.656,-75.648,169.809,34.075,156.427
C05421=1045.638,-30.407,-75.662,169.811,34.075,156.427
C05422=1045.645,-30.157,-75.675,169.813,34.077,156.428
C05423=1045.651,-29.908,-75.688,169.815,34.078,156.428
C05424=1045.658,-29.658,-75.702,169.817,34.079,156.428
C05425=1045.664,-29.408,-75.715,169.819,34.080,156.428
C05426=1045.671,-29.159,-75.729,169.821,34.082,156.428
